C03663=1150.971,190.773,-61.352,-178.173,7.203,148.817
C03664=1150.967,191.022,-61.376,-178.171,7.205,148.817
C03665=1150.962,191.271,-61.399,-178.168,7.208,148.817
C03666=1150.958,191.521,-61.423,-178.165,7.210,148.817
C03667=1150.954,191.769,-61.447,-178.162,7.213,148.816
C03668=1150.949,192.018,-61.470,-178.160,7.214,148.816
C03669=1150.944,192.267,-61.493,-178.157,7.217,148.816
C03670=1150.940,192.516,-61.518,-178.154,7.219,148.816
C03671=1150.935,192.765,-61.541,-178.151,7.222,148.815
C03672=1150.931,193.013,-61.565,-178.149,7.224,148.815
C03673=1150.926,193.262,-61.588,-178.145,7.226,148.815
C03674=1150.921,193.511,-61.612,-178.143,7.228,148.815
C03675=1150.917,193.759,-61.636,-178.140,7.231,148.814
C03676=1150.912,194.008,-61.659,-178.138,7.233,148.814
C03677=1150.907,194.257,-61.684,-178.134,7.235,148.814
C03678=1150.902,194.506,-61.707,-178.132,7.238,148.814
C03679=1150.898,194.755,-61.731,-178.129,7.240,148.813
C03680=1150.893,195.004,-61.755,-178.127,7.242,148.813
C03681=1150.889,195.252,-61.779,-178.123,7.245,148.813
C03682=1150.884,195.501,-61.802,-178.121,7.247,148.813
C03683=1150.880,195.750,-61.826,-178.118,7.249,148.812
C03684=1150.876,195.999,-61.850,-178.115,7.251,148.812
C03685=1150.871,196.248,-61.874,-178.112,7.254,148.812
C03686=1150.866,196.497,-61.898,-178.110,7.256,148.812
C03687=1150.862,196.745,-61.922,-178.107,7.259,148.812
C03688=1150.857,196.994,-61.945,-178.104,7.261,148.811
C03689=1150.852,197.243,-61.969,-178.101,7.263,148.811
C03690=1150.848,197.491,-61.993,-178.098,7.266,148.811
C03691=1150.843,197.741,-62.018,-178.096,7.268,148.811
C03692=1150.839,197.990,-62.042,-178.093,7.271,148.810
C03693=1150.834,198.238,-62.066,-178.090,7.273,148.810
C03694=1150.830,198.487,-62.089,-178.087,7.275,148.810
C03695=1150.825,198.736,-62.113,-178.085,7.277,148.810
C03696=1150.820,198.984,-62.138,-178.082,7.280,148.809
C03697=1150.816,199.234,-62.162,-178.079,7.282,148.809
C03698=1150.812,199.482,-62.186,-178.076,7.285,148.809
C03699=1150.807,199.731,-62.210,-178.074,7.287,148.809
C03700=1150.802,199.980,-62.235,-178.071,7.289,148.808
C03701=1150.797,200.229,-62.258,-178.068,7.292,148.808
C03702=1150.794,200.478,-62.282,-178.065,7.294,148.808
C03703=1150.789,200.726,-62.307,-178.062,7.297,148.808
C03704=1150.784,200.975,-62.331,-178.060,7.299,148.808
C03705=1150.779,201.224,-62.354,-178.057,7.302,148.807
C03706=1150.775,201.472,-62.379,-178.054,7.303,148.807
C03707=1150.770,201.722,-62.404,-178.052,7.306,148.807
C03708=1150.766,201.970,-62.428,-178.049,7.308,148.807
C03709=1150.762,202.219,-62.452,-178.046,7.311,148.807
C03710=1150.757,202.467,-62.476,-178.043,7.314,148.806
C03711=1150.753,202.716,-62.501,-178.041,7.316,148.806
C03712=1150.748,202.965,-62.524,-178.038,7.319,148.806
C03713=1150.743,203.214,-62.549,-178.035,7.320,148.806
C03714=1150.739,203.463,-62.573,-178.032,7.323,148.805
C03715=1150.734,203.712,-62.598,-178.030,7.325,148.805
C03716=1150.730,203.960,-62.622,-178.027,7.328,148.805
C03717=1150.725,204.209,-62.646,-178.024,7.330,148.805
C03718=1150.721,204.458,-62.671,-178.021,7.333,148.805
C03719=1150.716,204.707,-62.695,-178.018,7.335,148.804
C03720=1150.711,204.955,-62.720,-178.016,7.337,148.804
C03721=1150.707,205.204,-62.744,-178.013,7.340,148.804
C03722=1150.702,205.453,-62.769,-178.010,7.343,148.804
C03723=1150.698,205.702,-62.793,-178.008,7.345,148.804
C03724=1150.693,205.950,-62.818,-178.004,7.347,148.803
C03725=1150.689,206.199,-62.842,-178.002,7.349,148.803
C03726=1150.684,206.448,-62.867,-177.999,7.352,148.803
C03727=1150.679,206.697,-62.891,-177.996,7.355,148.803
C03728=1150.675,206.946,-62.916,-177.993,7.357,148.802
C03729=1150.670,207.194,-62.940,-177.991,7.360,148.802
C03730=1150.666,207.443,-62.965,-177.988,7.362,148.802
C03731=1150.662,207.692,-62.990,-177.985,7.364,148.802
C03732=1150.657,207.940,-63.015,-177.982,7.367,148.802
C03733=1150.652,208.189,-63.039,-177.980,7.369,148.801
C03734=1150.648,208.438,-63.064,-177.977,7.372,148.801
C03735=1150.643,208.687,-63.088,-177.974,7.374,148.801
C03736=1150.639,208.936,-63.113,-177.971,7.377,148.801
C03737=1150.634,209.184,-63.138,-177.969,7.379,148.801
C03738=1150.629,209.454,-63.165,-177.965,7.382,148.800
C03739=1150.624,209.725,-63.192,-177.963,7.385,148.800
C03740=1150.619,209.995,-63.219,-177.960,7.387,148.800
C03741=1150.615,210.266,-63.246,-177.957,7.390,148.800
C03742=1150.610,210.515,-63.270,-177.954,7.392,148.800
C03743=1150.606,210.764,-63.295,-177.951,7.395,148.799
C03744=1150.601,211.013,-63.319,-177.948,7.397,148.799
C03745=1150.597,211.261,-63.345,-177.946,7.400,148.799
C03746=1150.592,211.510,-63.369,-177.943,7.403,148.799
C03747=1150.587,211.759,-63.394,-177.940,7.405,148.799
C03748=1150.583,212.007,-63.419,-177.937,7.407,148.798
C03749=1150.578,212.256,-63.444,-177.935,7.409,148.798
C03750=1150.574,212.505,-63.469,-177.932,7.412,148.798
C03751=1150.569,212.753,-63.494,-177.929,7.415,148.798
C03752=1150.565,213.003,-63.519,-177.926,7.417,148.798
C03753=1150.560,213.251,-63.544,-177.924,7.420,148.797
C03754=1150.556,213.500,-63.569,-177.921,7.423,148.797
C03755=1150.552,213.748,-63.594,-177.918,7.424,148.797
C03756=1150.547,213.997,-63.619,-177.915,7.427,148.797
C03757=1150.542,214.246,-63.644,-177.912,7.430,148.797
C03758=1150.538,214.495,-63.669,-177.910,7.432,148.797
C03759=1150.533,214.743,-63.693,-177.907,7.435,148.796
C03760=1150.529,214.992,-63.719,-177.904,7.437,148.796
C03761=1150.524,215.241,-63.744,-177.902,7.440,148.796
C03762=1150.520,215.490,-63.770,-177.899,7.443,148.796
C03763=1150.515,215.738,-63.794,-177.895,7.445,148.796
C03764=1150.511,215.987,-63.819,-177.893,7.447,148.795
C03765=1150.506,216.235,-63.845,-177.890,7.450,148.795
C03766=1150.502,216.484,-63.870,-177.887,7.453,148.795
C03767=1150.497,216.732,-63.895,-177.885,7.455,148.795
C03768=1150.492,216.982,-63.920,-177.882,7.458,148.795
C03769=1150.488,217.230,-63.945,-177.879,7.460,148.795
C03770=1150.484,217.478,-63.971,-177.877,7.462,148.794
C03771=1150.480,217.728,-63.996,-177.874,7.465,148.794
C03772=1150.475,217.976,-64.021,-177.871,7.468,148.794
C03773=1150.471,218.225,-64.047,-177.868,7.470,148.794
C03774=1150.465,218.474,-64.072,-177.866,7.473,148.794
C03775=1150.461,218.722,-64.097,-177.862,7.476,148.793
C03776=1150.457,218.971,-64.123,-177.860,7.478,148.793
C03777=1150.452,219.220,-64.148,-177.857,7.481,148.793
C03778=1150.448,219.468,-64.173,-177.855,7.483,148.793
C03779=1150.444,219.716,-64.198,-177.851,7.486,148.793
C03780=1150.439,219.965,-64.224,-177.849,7.488,148.793
C03781=1150.435,220.215,-64.249,-177.846,7.491,148.793
C03782=1150.430,220.463,-64.275,-177.843,7.494,148.792
C03783=1150.426,220.712,-64.300,-177.840,7.497,148.792
C03784=1150.421,220.960,-64.326,-177.838,7.499,148.792
C03785=1150.417,221.209,-64.351,-177.835,7.501,148.792
C03786=1150.412,221.458,-64.376,-177.832,7.504,148.792
C03787=1150.407,221.706,-64.402,-177.830,7.506,148.792
C03788=1150.403,221.955,-64.428,-177.827,7.509,148.792
C03789=1150.399,222.204,-64.453,-177.824,7.512,148.791
C03790=1150.394,222.452,-64.479,-177.821,7.515,148.791
C03791=1150.390,222.701,-64.504,-177.819,7.517,148.791
C03792=1150.386,222.949,-64.530,-177.816,7.519,148.791
C03793=1150.381,223.197,-64.556,-177.813,7.522,148.791
C03794=1150.377,223.446,-64.581,-177.811,7.524,148.790
C03795=1150.372,223.695,-64.607,-177.808,7.527,148.790
C03796=1150.367,223.944,-64.633,-177.805,7.530,148.790
C03797=1150.362,224.193,-64.658,-177.802,7.533,148.790
C03798=1150.358,224.442,-64.684,-177.800,7.535,148.790
C03799=1150.354,224.691,-64.710,-177.797,7.538,148.790
C03800=1150.349,224.939,-64.735,-177.793,7.540,148.789
C03801=1150.345,225.187,-64.761,-177.791,7.543,148.789
C03802=1150.341,225.436,-64.787,-177.788,7.545,148.789
C03803=1150.337,225.684,-64.813,-177.786,7.548,148.789
C03804=1150.332,225.933,-64.838,-177.782,7.551,148.789
C03805=1150.327,226.182,-64.865,-177.780,7.554,148.789
C03806=1150.323,226.430,-64.890,-177.777,7.556,148.789
C03807=1150.318,226.679,-64.916,-177.775,7.559,148.789
C03808=1150.314,226.927,-64.942,-177.771,7.562,148.788
C03809=1150.309,227.176,-64.967,-177.769,7.564,148.788
C03810=1150.304,227.425,-64.994,-177.766,7.567,148.788
C03811=1150.300,227.673,-65.020,-177.764,7.569,148.788
C03812=1150.296,227.922,-65.046,-177.760,7.572,148.788
C03813=1150.291,228.170,-65.071,-177.758,7.575,148.788
C03814=1150.287,228.419,-65.097,-177.755,7.578,148.788
C03815=1150.282,228.668,-65.123,-177.753,7.580,148.787
C03816=1150.278,228.917,-65.149,-177.750,7.583,148.787
C03817=1150.273,229.165,-65.175,-177.747,7.586,148.787
C03818=1150.269,229.413,-65.201,-177.744,7.588,148.787
C03819=1150.264,229.663,-65.227,-177.742,7.591,148.787
C03820=1150.260,229.911,-65.254,-177.739,7.593,148.787
C03821=1150.256,230.160,-65.280,-177.736,7.596,148.786
C03822=1150.251,230.409,-65.306,-177.733,7.599,148.786
C03823=1150.246,230.657,-65.331,-177.730,7.602,148.786
C03824=1150.242,230.905,-65.358,-177.728,7.604,148.786
C03825=1150.237,231.154,-65.384,-177.725,7.607,148.786
C03826=1150.233,231.403,-65.410,-177.722,7.610,148.786
C03827=1150.229,231.651,-65.436,-177.719,7.612,148.786
C03828=1150.224,231.900,-65.463,-177.716,7.615,148.786
C03829=1150.220,232.148,-65.489,-177.714,7.618,148.785
C03830=1150.216,232.396,-65.514,-177.711,7.620,148.785
C03831=1150.211,232.646,-65.541,-177.708,7.623,148.785
C03832=1150.207,232.894,-65.567,-177.705,7.626,148.785
C03833=1150.202,233.143,-65.594,-177.702,7.629,148.785
C03834=1150.198,233.391,-65.620,-177.700,7.631,148.785
C03835=1150.194,233.640,-65.646,-177.697,7.634,148.785
C03836=1150.189,233.888,-65.673,-177.695,7.637,148.785
C03837=1150.185,234.137,-65.699,-177.691,7.639,148.784
C03838=1150.180,234.386,-65.726,-177.688,7.642,148.784
C03839=1150.176,234.634,-65.751,-177.686,7.644,148.784
C03840=1150.171,234.882,-65.778,-177.684,7.647,148.784
C03841=1150.166,235.131,-65.804,-177.681,7.650,148.784
C03842=1150.162,235.403,-65.834,-177.678,7.653,148.784
C03843=1150.157,235.675,-65.862,-177.675,7.656,148.784
C03844=1150.152,235.947,-65.891,-177.671,7.660,148.784
C03845=1150.148,236.218,-65.920,-177.669,7.663,148.784
C03846=1150.143,236.467,-65.947,-177.666,7.665,148.783
C03847=1150.139,236.715,-65.973,-177.663,7.667,148.783
C03848=1150.134,236.964,-66.000,-177.660,7.670,148.783
C03849=1150.130,237.213,-66.025,-177.658,7.673,148.783
C03850=1150.125,237.461,-66.052,-177.655,7.676,148.783
C03851=1150.121,237.710,-66.080,-177.652,7.679,148.783
C03852=1150.117,237.958,-66.106,-177.649,7.682,148.783
C03853=1150.112,238.207,-66.132,-177.646,7.685,148.783
C03854=1150.108,238.455,-66.159,-177.644,7.687,148.782
C03855=1150.103,238.704,-66.186,-177.641,7.689,148.782
C03856=1150.099,238.952,-66.212,-177.638,7.692,148.782
C03857=1150.094,239.201,-66.239,-177.635,7.695,148.782
C03858=1150.090,239.449,-66.266,-177.633,7.698,148.782
C03859=1150.086,239.698,-66.292,-177.630,7.701,148.782
C03860=1150.081,239.946,-66.319,-177.628,7.703,148.782
C03861=1150.076,240.195,-66.346,-177.625,7.706,148.782
C03862=1150.072,240.443,-66.372,-177.622,7.709,148.782
C03863=1150.067,240.692,-66.399,-177.619,7.712,148.781
C03864=1150.063,240.940,-66.426,-177.616,7.715,148.781
C03865=1150.059,241.189,-66.453,-177.613,7.718,148.781
C03866=1150.054,241.437,-66.480,-177.610,7.721,148.781
C03867=1150.050,241.686,-66.507,-177.608,7.723,148.781
C03868=1150.046,241.935,-66.534,-177.605,7.726,148.781
C03869=1150.041,242.184,-66.560,-177.603,7.728,148.781
C03870=1150.037,242.432,-66.587,-177.600,7.731,148.781
C03871=1150.033,242.680,-66.614,-177.597,7.734,148.781
C03872=1150.028,242.929,-66.641,-177.594,7.737,148.781
C03873=1150.023,243.177,-66.668,-177.591,7.740,148.780
C03874=1150.019,243.426,-66.695,-177.588,7.743,148.780
C03875=1150.015,243.674,-66.721,-177.585,7.746,148.780
C03876=1150.011,243.923,-66.749,-177.583,7.748,148.780
C03877=1150.006,244.172,-66.776,-177.580,7.751,148.780
C03878=1150.001,244.420,-66.803,-177.578,7.754,148.780
C03879=1149.997,244.669,-66.830,-177.575,7.757,148.780
C03880=1149.993,244.916,-66.857,-177.572,7.760,148.780
C03881=1149.988,245.165,-66.884,-177.569,7.763,148.780
C03882=1149.984,245.413,-66.911,-177.567,7.765,148.780
C03883=1149.980,245.662,-66.939,-177.564,7.768,148.780
C03884=1149.975,245.911,-66.966,-177.561,7.771,148.780
C03885=1149.970,246.159,-66.993,-177.559,7.773,148.779
C03886=1149.967,246.408,-67.019,-177.556,7.776,148.779
C03887=1149.962,246.656,-67.046,-177.553,7.779,148.779
C03888=1149.958,246.904,-67.074,-177.550,7.782,148.779
C03889=1149.953,247.153,-67.101,-177.547,7.785,148.779
C03890=1149.949,247.402,-67.128,-177.544,7.788,148.779
C03891=1149.944,247.650,-67.155,-177.542,7.791,148.779
C03892=1149.940,247.899,-67.183,-177.539,7.794,148.779
C03893=1149.936,248.147,-67.211,-177.536,7.797,148.779
C03894=1149.931,248.396,-67.238,-177.533,7.799,148.779
C03895=1149.926,248.644,-67.265,-177.531,7.802,148.778
C03896=1149.923,248.892,-67.291,-177.528,7.804,148.778
C03897=1149.918,249.140,-67.319,-177.526,7.807,148.778
C03898=1149.914,249.389,-67.346,-177.523,7.810,148.778
C03899=1149.909,249.638,-67.374,-177.520,7.813,148.778
C03900=1149.905,249.886,-67.401,-177.517,7.816,148.778
C03901=1149.900,250.134,-67.428,-177.514,7.819,148.778
C03902=1149.896,250.384,-67.456,-177.512,7.822,148.778
C03903=1149.892,250.631,-67.484,-177.509,7.825,148.778
C03904=1149.887,250.880,-67.511,-177.506,7.828,148.778
C03905=1149.884,251.128,-67.539,-177.503,7.831,148.778
C03906=1149.879,251.377,-67.566,-177.500,7.834,148.778
C03907=1149.875,251.625,-67.594,-177.498,7.837,148.778
C03908=1149.870,251.873,-67.621,-177.495,7.840,148.778
C03909=1149.865,252.123,-67.649,-177.493,7.842,148.777
C03910=1149.861,252.371,-67.676,-177.490,7.845,148.777
C03911=1149.856,252.619,-67.704,-177.487,7.848,148.777
C03912=1149.852,252.868,-67.732,-177.484,7.851,148.777
C03913=1149.848,253.116,-67.759,-177.482,7.854,148.777
C03914=1149.843,253.364,-67.787,-177.479,7.856,148.777
C03915=1149.839,253.613,-67.814,-177.476,7.859,148.777
C03916=1149.835,253.861,-67.842,-177.473,7.862,148.777
C03917=1149.831,254.109,-67.870,-177.470,7.865,148.777
C03918=1149.827,254.358,-67.897,-177.468,7.868,148.777
C03919=1149.822,254.607,-67.925,-177.465,7.871,148.777
C03920=1149.817,254.855,-67.952,-177.462,7.874,148.777
C03921=1149.813,255.104,-67.981,-177.459,7.877,148.777
C03922=1149.809,255.351,-68.008,-177.457,7.880,148.777
C03923=1149.805,255.601,-68.036,-177.454,7.883,148.777
C03924=1149.800,255.849,-68.064,-177.451,7.886,148.777
C03925=1149.795,256.097,-68.092,-177.449,7.889,148.777
C03926=1149.791,256.346,-68.119,-177.446,7.892,148.777
C03927=1149.787,256.594,-68.147,-177.443,7.895,148.776
C03928=1149.783,256.842,-68.175,-177.440,7.898,148.776
C03929=1149.778,257.091,-68.203,-177.438,7.901,148.776
C03930=1149.773,257.339,-68.231,-177.435,7.904,148.776
C03931=1149.770,257.588,-68.259,-177.433,7.906,148.776
C03932=1149.765,257.835,-68.287,-177.430,7.909,148.776
C03933=1149.760,258.085,-68.315,-177.427,7.912,148.776
C03934=1149.756,258.333,-68.342,-177.424,7.915,148.776
C03935=1149.752,258.581,-68.371,-177.421,7.918,148.776
C03936=1149.748,258.829,-68.398,-177.419,7.921,148.776
C03937=1149.743,259.078,-68.427,-177.416,7.923,148.776
C03938=1149.739,259.326,-68.455,-177.414,7.927,148.776
C03939=1149.735,259.575,-68.482,-177.411,7.930,148.776
C03940=1149.730,259.823,-68.511,-177.408,7.933,148.776
C03941=1149.726,260.071,-68.538,-177.405,7.936,148.776
C03942=1149.722,260.320,-68.567,-177.402,7.938,148.776
C03943=1149.717,260.568,-68.595,-177.400,7.941,148.776
C03944=1149.713,260.817,-68.623,-177.397,7.944,148.776
C03945=1149.709,261.065,-68.651,-177.394,7.947,148.776
C03946=1149.703,261.338,-68.682,-177.391,7.951,148.776
C03947=1149.699,261.612,-68.713,-177.388,7.954,148.775
C03948=1149.695,261.886,-68.744,-177.385,7.957,148.775
C03949=1149.690,262.159,-68.776,-177.382,7.961,148.775
C03950=1149.685,262.406,-68.804,-177.379,7.964,148.775
C03951=1149.681,262.655,-68.832,-177.377,7.967,148.775
C03952=1149.676,262.903,-68.860,-177.374,7.970,148.775
C03953=1149.673,263.152,-68.888,-177.371,7.973,148.775
C03954=1149.667,263.400,-68.917,-177.368,7.976,148.775
C03955=1149.664,263.649,-68.945,-177.366,7.979,148.775
C03956=1149.659,263.897,-68.973,-177.363,7.982,148.775
C03957=1149.655,264.145,-69.001,-177.360,7.984,148.775
C03958=1149.650,264.394,-69.030,-177.357,7.987,148.775
C03959=1149.646,264.642,-69.058,-177.355,7.991,148.775
C03960=1149.642,264.890,-69.087,-177.352,7.994,148.775
C03961=1149.638,265.138,-69.115,-177.349,7.997,148.775
C03962=1149.633,265.387,-69.144,-177.347,7.999,148.775
C03963=1149.629,265.636,-69.172,-177.344,8.002,148.775
C03964=1149.624,265.884,-69.200,-177.341,8.005,148.775
C03965=1149.621,266.132,-69.229,-177.339,8.009,148.775
C03966=1149.616,266.380,-69.258,-177.336,8.012,148.775
C03967=1149.611,266.629,-69.286,-177.333,8.014,148.775
C03968=1149.607,266.878,-69.314,-177.330,8.017,148.775
C03969=1149.603,267.125,-69.343,-177.328,8.020,148.775
C03970=1149.599,267.374,-69.372,-177.325,8.023,148.775
C03971=1149.594,267.622,-69.400,-177.323,8.027,148.775
C03972=1149.590,267.870,-69.429,-177.320,8.029,148.775
C03973=1149.586,268.119,-69.458,-177.317,8.032,148.775
C03974=1149.581,268.367,-69.486,-177.314,8.035,148.775
C03975=1149.577,268.615,-69.515,-177.311,8.038,148.775
C03976=1149.573,268.864,-69.544,-177.309,8.042,148.775
C03977=1149.568,269.112,-69.572,-177.306,8.045,148.775
C03978=1149.564,269.360,-69.601,-177.303,8.048,148.775
C03979=1149.560,269.609,-69.630,-177.300,8.051,148.775
C03980=1149.555,269.856,-69.659,-177.297,8.054,148.775
C03981=1149.551,270.105,-69.687,-177.295,8.057,148.775
C03982=1149.547,270.354,-69.715,-177.292,8.060,148.775
C03983=1149.543,270.602,-69.745,-177.290,8.063,148.775
C03984=1149.538,270.850,-69.773,-177.287,8.066,148.775
C03985=1149.534,271.098,-69.802,-177.284,8.069,148.775
C03986=1149.530,271.347,-69.831,-177.282,8.072,148.775
C03987=1149.525,271.595,-69.860,-177.279,8.075,148.775
C03988=1149.520,271.844,-69.889,-177.276,8.078,148.775
C03989=1149.517,272.091,-69.918,-177.273,8.081,148.775
C03990=1149.513,272.340,-69.947,-177.271,8.084,148.775
C03991=1149.508,272.588,-69.975,-177.268,8.087,148.775
C03992=1149.503,272.836,-70.005,-177.265,8.090,148.775
C03993=1149.499,273.085,-70.034,-177.262,8.094,148.775
C03994=1149.496,273.333,-70.062,-177.260,8.097,148.775
C03995=1149.491,273.581,-70.092,-177.257,8.100,148.775
C03996=1149.486,273.830,-70.120,-177.254,8.103,148.775
C03997=1149.482,274.078,-70.150,-177.251,8.106,148.775
C03998=1149.478,274.326,-70.179,-177.249,8.109,148.775
C03999=1149.473,274.575,-70.208,-177.246,8.112,148.775
C04000=1149.469,274.822,-70.236,-177.244,8.115,148.775
C04001=1149.465,275.070,-70.266,-177.241,8.118,148.775
C04002=1149.461,275.319,-70.295,-177.238,8.122,148.775
C04003=1149.457,275.568,-70.324,-177.236,8.125,148.775
C04004=1149.452,275.816,-70.354,-177.233,8.127,148.775
C04005=1149.448,276.064,-70.383,-177.230,8.130,148.775
C04006=1149.443,276.312,-70.412,-177.227,8.134,148.775
C04007=1149.439,276.561,-70.441,-177.224,8.137,148.775
C04008=1149.435,276.809,-70.470,-177.222,8.140,148.775
C04009=1149.431,277.057,-70.499,-177.219,8.144,148.775
C04010=1149.427,277.305,-70.529,-177.217,8.147,148.775
C04011=1149.423,277.553,-70.558,-177.214,8.149,148.775
C04012=1149.418,277.801,-70.587,-177.212,8.153,148.775
C04013=1149.414,278.050,-70.616,-177.209,8.156,148.775
C04014=1149.409,278.298,-70.645,-177.206,8.159,148.775
C04015=1149.405,278.546,-70.675,-177.203,8.162,148.775
C04016=1149.401,278.795,-70.704,-177.200,8.166,148.775
C04017=1149.397,279.043,-70.734,-177.198,8.169,148.775
C04018=1149.393,279.291,-70.763,-177.195,8.172,148.775
C04019=1149.389,279.539,-70.793,-177.192,8.175,148.775
C04020=1149.384,279.788,-70.822,-177.190,8.178,148.775
C04021=1149.380,280.036,-70.851,-177.187,8.181,148.775
C04022=1149.375,280.284,-70.881,-177.185,8.184,148.775
C04023=1149.371,280.532,-70.910,-177.182,8.187,148.775
C04024=1149.366,280.780,-70.940,-177.179,8.190,148.775
C04025=1149.362,281.029,-70.970,-177.176,8.194,148.775
C04026=1149.358,281.277,-70.999,-177.173,8.197,148.775
C04027=1149.354,281.525,-71.028,-177.171,8.200,148.775
C04028=1149.350,281.773,-71.058,-177.168,8.203,148.775
C04029=1149.345,282.022,-71.087,-177.165,8.206,148.775
C04030=1149.342,282.269,-71.118,-177.163,8.209,148.775
C04031=1149.337,282.518,-71.147,-177.160,8.212,148.775
C04032=1149.332,282.766,-71.177,-177.158,8.215,148.775
C04033=1149.328,283.014,-71.206,-177.155,8.219,148.776
C04034=1149.324,283.263,-71.236,-177.152,8.222,148.776
C04035=1149.320,283.511,-71.265,-177.149,8.225,148.776
C04036=1149.316,283.759,-71.295,-177.147,8.228,148.776
C04037=1149.312,284.007,-71.325,-177.144,8.231,148.776
C04038=1149.307,284.255,-71.355,-177.142,8.235,148.776
C04039=1149.303,284.504,-71.384,-177.139,8.238,148.776
C04040=1149.299,284.752,-71.414,-177.136,8.241,148.776
C04041=1149.295,285.000,-71.444,-177.133,8.245,148.776
C04042=1149.290,285.248,-71.474,-177.130,8.248,148.776
C04043=1149.286,285.497,-71.504,-177.128,8.251,148.776
C04044=1149.282,285.744,-71.534,-177.125,8.254,148.776
C04045=1149.277,285.992,-71.563,-177.123,8.257,148.776
C04046=1149.273,286.241,-71.593,-177.120,8.260,148.776
C04047=1149.269,286.489,-71.623,-177.117,8.264,148.776
C04048=1149.265,286.737,-71.653,-177.115,8.267,148.776
C04049=1149.260,286.985,-71.682,-177.112,8.270,148.776
C04050=1149.256,287.261,-71.717,-177.109,8.273,148.776
C04051=1149.251,287.536,-71.749,-177.106,8.277,148.776
C04052=1149.246,287.811,-71.783,-177.103,8.281,148.776
C04053=1149.241,288.086,-71.816,-177.100,8.284,148.776
C04054=1149.238,288.335,-71.846,-177.097,8.288,148.777
C04055=1149.233,288.583,-71.876,-177.094,8.291,148.777
C04056=1149.229,288.831,-71.906,-177.092,8.294,148.777
C04057=1149.224,289.079,-71.937,-177.089,8.297,148.777
C04058=1149.220,289.327,-71.966,-177.087,8.300,148.777
C04059=1149.216,289.575,-71.996,-177.084,8.303,148.777
C04060=1149.211,289.824,-72.026,-177.081,8.307,148.777
C04061=1149.207,290.071,-72.057,-177.078,8.310,148.777
C04062=1149.203,290.320,-72.087,-177.076,8.313,148.777
C04063=1149.199,290.568,-72.117,-177.073,8.316,148.777
C04064=1149.195,290.816,-72.147,-177.071,8.319,148.777
C04065=1149.191,291.064,-72.177,-177.068,8.323,148.777
C04066=1149.187,291.312,-72.207,-177.065,8.326,148.777
C04067=1149.182,291.561,-72.238,-177.063,8.330,148.777
C04068=1149.178,291.808,-72.268,-177.060,8.333,148.777
C04069=1149.174,292.057,-72.299,-177.058,8.336,148.778
C04070=1149.170,292.305,-72.328,-177.055,8.339,148.777
C04071=1149.165,292.553,-72.359,-177.052,8.343,148.778
C04072=1149.161,292.801,-72.389,-177.049,8.346,148.778
C04073=1149.156,293.049,-72.419,-177.047,8.349,148.778
C04074=1149.153,293.298,-72.450,-177.044,8.352,148.778
C04075=1149.148,293.546,-72.481,-177.042,8.355,148.778
C04076=1149.144,293.793,-72.511,-177.038,8.359,148.778
C04077=1149.140,294.042,-72.541,-177.036,8.362,148.778
C04078=1149.136,294.290,-72.571,-177.033,8.365,148.778
C04079=1149.132,294.538,-72.602,-177.031,8.369,148.778
C04080=1149.128,294.786,-72.632,-177.029,8.372,148.778
C04081=1149.123,295.034,-72.663,-177.025,8.376,148.778
C04082=1149.119,295.282,-72.694,-177.023,8.379,148.779
C04083=1149.115,295.531,-72.724,-177.020,8.382,148.779
C04084=1149.110,295.779,-72.754,-177.018,8.385,148.779
C04085=1149.106,296.026,-72.785,-177.015,8.388,148.779
C04086=1149.102,296.275,-72.816,-177.012,8.392,148.779
C04087=1149.098,296.523,-72.846,-177.009,8.395,148.779
C04088=1149.094,296.771,-72.877,-177.007,8.398,148.779
C04089=1149.089,297.019,-72.907,-177.004,8.401,148.779
C04090=1149.085,297.267,-72.938,-177.002,8.404,148.779
C04091=1149.081,297.515,-72.969,-176.999,8.409,148.779
C04092=1149.077,297.763,-72.999,-176.996,8.412,148.779
C04093=1149.073,298.011,-73.031,-176.994,8.415,148.780
C04094=1149.069,298.259,-73.061,-176.991,8.418,148.780
C04095=1149.064,298.507,-73.091,-176.988,8.422,148.780
C04096=1149.060,298.756,-73.123,-176.986,8.425,148.780
C04097=1149.056,299.003,-73.153,-176.983,8.428,148.780
C04098=1149.052,299.251,-73.184,-176.981,8.431,148.780
C04099=1149.048,299.500,-73.215,-176.978,8.435,148.780
C04100=1149.043,299.748,-73.245,-176.975,8.438,148.780
C04101=1149.039,299.996,-73.276,-176.972,8.441,148.780
C04102=1149.035,300.244,-73.307,-176.970,8.445,148.780
C04103=1149.031,300.492,-73.338,-176.968,8.448,148.781
C04104=1149.026,300.740,-73.369,-176.964,8.452,148.781
C04105=1149.022,300.988,-73.400,-176.962,8.455,148.781
C04106=1149.019,301.236,-73.430,-176.959,8.458,148.781
C04107=1149.014,301.484,-73.461,-176.957,8.461,148.781
C04108=1149.010,301.732,-73.492,-176.954,8.465,148.781
C04109=1149.006,301.980,-73.524,-176.951,8.468,148.781
C04110=1149.002,302.228,-73.555,-176.949,8.471,148.781
C04111=1148.997,302.476,-73.586,-176.947,8.475,148.781
C04112=1148.993,302.724,-73.616,-176.943,8.478,148.781
C04113=1148.989,302.972,-73.648,-176.941,8.482,148.782
C04114=1148.985,303.220,-73.678,-176.939,8.485,148.782
C04115=1148.981,303.469,-73.709,-176.936,8.488,148.782
C04116=1148.976,303.716,-73.741,-176.933,8.492,148.782
C04117=1148.972,303.964,-73.772,-176.931,8.495,148.782
C04118=1148.968,304.213,-73.803,-176.928,8.498,148.782
C04119=1148.964,304.460,-73.834,-176.925,8.502,148.782
C04120=1148.960,304.709,-73.865,-176.923,8.506,148.783
C04121=1148.955,304.957,-73.896,-176.920,8.508,148.783
C04122=1148.951,305.205,-73.928,-176.918,8.512,148.783
C04123=1148.947,305.453,-73.959,-176.915,8.516,148.783
C04124=1148.943,305.701,-73.991,-176.912,8.519,148.783
C04125=1148.938,305.949,-74.021,-176.910,8.522,148.783
C04126=1148.935,306.197,-74.053,-176.907,8.525,148.783
C04127=1148.930,306.445,-74.084,-176.904,8.529,148.783
C04128=1148.926,306.693,-74.116,-176.902,8.532,148.783
C04129=1148.922,306.941,-74.147,-176.899,8.536,148.784
C04130=1148.918,307.189,-74.178,-176.896,8.539,148.784
C04131=1148.913,307.437,-74.209,-176.894,8.543,148.784
C04132=1148.910,307.685,-74.241,-176.891,8.546,148.784
C04133=1148.905,307.933,-74.272,-176.889,8.549,148.784
C04134=1148.901,308.181,-74.304,-176.886,8.553,148.784
C04135=1148.897,308.429,-74.334,-176.883,8.556,148.784
C04136=1148.893,308.677,-74.366,-176.881,8.560,148.785
C04137=1148.889,308.924,-74.398,-176.878,8.563,148.785
C04138=1148.885,309.173,-74.429,-176.875,8.567,148.785
C04139=1148.880,309.420,-74.460,-176.873,8.570,148.785
C04140=1148.877,309.668,-74.492,-176.871,8.573,148.785
C04141=1148.871,309.916,-74.524,-176.867,8.577,148.785
C04142=1148.868,310.164,-74.555,-176.865,8.580,148.785
C04143=1148.864,310.412,-74.587,-176.863,8.583,148.786
C04144=1148.859,310.660,-74.618,-176.860,8.587,148.786
C04145=1148.856,310.908,-74.650,-176.857,8.590,148.786
C04146=1148.851,311.156,-74.681,-176.855,8.594,148.786
C04147=1148.848,311.404,-74.713,-176.852,8.598,148.786
C04148=1148.842,311.652,-74.745,-176.849,8.601,148.786
C04149=1148.838,311.900,-74.776,-176.847,8.604,148.786
C04150=1148.835,312.148,-74.808,-176.844,8.608,148.787
C04151=1148.830,312.395,-74.840,-176.841,8.611,148.787
C04152=1148.827,312.643,-74.872,-176.839,8.615,148.787
C04153=1148.822,312.892,-74.904,-176.837,8.618,148.787
C04154=1148.817,313.169,-74.939,-176.833,8.622,148.787
C04155=1148.813,313.447,-74.974,-176.831,8.626,148.787
C04156=1148.808,313.724,-75.010,-176.828,8.630,148.788
C04157=1148.803,314.002,-75.046,-176.825,8.634,148.788
C04158=1148.800,314.250,-75.078,-176.822,8.637,148.788
C04159=1148.795,314.498,-75.109,-176.819,8.641,148.788
C04160=1148.791,314.746,-75.142,-176.817,8.644,148.788
C04161=1148.787,314.994,-75.174,-176.814,8.648,148.788
C04162=1148.783,315.241,-75.205,-176.811,8.652,148.789
C04163=1148.779,315.489,-75.237,-176.809,8.655,148.789
C04164=1148.775,315.738,-75.269,-176.806,8.658,148.789
C04165=1148.770,315.985,-75.301,-176.803,8.662,148.789
C04166=1148.767,316.233,-75.333,-176.801,8.665,148.789
C04167=1148.762,316.481,-75.365,-176.799,8.668,148.789
C04168=1148.759,316.729,-75.397,-176.796,8.673,148.790
C04169=1148.754,316.977,-75.429,-176.794,8.676,148.790
C04170=1148.750,317.225,-75.461,-176.791,8.679,148.790
C04171=1148.746,317.473,-75.493,-176.788,8.683,148.790
C04172=1148.742,317.721,-75.525,-176.786,8.686,148.790
C04173=1148.737,317.969,-75.557,-176.783,8.689,148.790
C04174=1148.733,318.217,-75.590,-176.780,8.693,148.791
C04175=1148.730,318.465,-75.622,-176.778,8.697,148.791
C04176=1148.726,318.713,-75.653,-176.776,8.700,148.791
C04177=1148.721,318.960,-75.686,-176.773,8.704,148.791
C04178=1148.717,319.208,-75.717,-176.770,8.707,148.791
C04179=1148.713,319.456,-75.751,-176.768,8.710,148.791
C04180=1148.709,319.704,-75.782,-176.765,8.714,148.792
C04181=1148.705,319.952,-75.815,-176.762,8.718,148.792
C04182=1148.701,320.200,-75.846,-176.760,8.722,148.792
C04183=1148.696,320.447,-75.879,-176.757,8.725,148.792
C04184=1148.693,320.696,-75.911,-176.755,8.728,148.792
C04185=1148.688,320.944,-75.944,-176.752,8.732,148.793
C04186=1148.685,321.191,-75.976,-176.750,8.736,148.793
C04187=1148.680,321.439,-76.008,-176.747,8.739,148.793
C04188=1148.676,321.687,-76.040,-176.744,8.743,148.793
C04189=1148.672,321.935,-76.073,-176.742,8.746,148.793
C04190=1148.668,322.183,-76.105,-176.739,8.750,148.793
C04191=1148.664,322.431,-76.138,-176.736,8.753,148.794
C04192=1148.660,322.679,-76.170,-176.734,8.757,148.794
C04193=1148.656,322.927,-76.203,-176.731,8.761,148.794
C04194=1148.651,323.174,-76.235,-176.729,8.764,148.794
C04195=1148.647,323.422,-76.267,-176.727,8.767,148.794
C04196=1148.643,323.670,-76.300,-176.724,8.771,148.795
C04197=1148.640,323.918,-76.332,-176.721,8.775,148.795
C04198=1148.636,324.165,-76.365,-176.718,8.779,148.795
C04199=1148.631,324.414,-76.398,-176.716,8.782,148.795
C04200=1148.628,324.661,-76.430,-176.714,8.785,148.795
C04201=1148.623,324.910,-76.463,-176.711,8.789,148.796
C04202=1148.618,325.157,-76.496,-176.709,8.793,148.796
C04203=1148.615,325.405,-76.528,-176.706,8.797,148.796
C04204=1148.611,325.652,-76.561,-176.703,8.800,148.796
C04205=1148.607,325.900,-76.594,-176.701,8.803,148.797
C04206=1148.603,326.148,-76.626,-176.698,8.807,148.797
C04207=1148.599,326.396,-76.659,-176.696,8.811,148.797
C04208=1148.594,326.644,-76.691,-176.693,8.815,148.797
C04209=1148.591,326.892,-76.724,-176.691,8.818,148.797
C04210=1148.587,327.139,-76.757,-176.688,8.822,148.798
C04211=1148.582,327.388,-76.789,-176.685,8.825,148.798
C04212=1148.578,327.635,-76.823,-176.683,8.829,148.798
C04213=1148.575,327.883,-76.855,-176.680,8.833,148.798
C04214=1148.571,328.131,-76.888,-176.678,8.836,148.798
C04215=1148.566,328.379,-76.921,-176.675,8.840,148.799
C04216=1148.562,328.627,-76.954,-176.673,8.843,148.799
C04217=1148.558,328.874,-76.987,-176.670,8.846,148.799
C04218=1148.554,329.122,-77.020,-176.667,8.851,148.799
C04219=1148.550,329.370,-77.052,-176.665,8.854,148.799
C04220=1148.546,329.618,-77.085,-176.662,8.858,148.800
C04221=1148.542,329.866,-77.118,-176.660,8.861,148.800
C04222=1148.538,330.113,-77.152,-176.657,8.865,148.800
C04223=1148.533,330.361,-77.185,-176.654,8.869,148.800
C04224=1148.529,330.609,-77.218,-176.652,8.872,148.801
C04225=1148.526,330.856,-77.250,-176.649,8.876,148.801
C04226=1148.521,331.105,-77.283,-176.647,8.879,148.801
C04227=1148.517,331.352,-77.316,-176.644,8.883,148.801
C04228=1148.513,331.600,-77.349,-176.642,8.887,148.801
C04229=1148.509,331.848,-77.382,-176.639,8.891,148.802
C04230=1148.505,332.095,-77.416,-176.637,8.894,148.802
C04231=1148.501,332.343,-77.449,-176.634,8.898,148.802
C04232=1148.497,332.591,-77.482,-176.632,8.902,148.803
C04233=1148.492,332.839,-77.515,-176.629,8.905,148.803
C04234=1148.488,333.086,-77.548,-176.626,8.909,148.803
C04235=1148.484,333.334,-77.581,-176.624,8.912,148.803
C04236=1148.480,333.582,-77.614,-176.621,8.916,148.803
C04237=1148.476,333.830,-77.648,-176.619,8.920,148.804
C04238=1148.472,334.078,-77.681,-176.616,8.924,148.804
C04239=1148.469,334.325,-77.715,-176.614,8.927,148.804
C04240=1148.464,334.573,-77.748,-176.611,8.931,148.804
C04241=1148.460,334.821,-77.781,-176.609,8.935,148.805
C04242=1148.456,335.068,-77.814,-176.606,8.939,148.805
C04243=1148.452,335.316,-77.848,-176.604,8.942,148.805
C04244=1148.448,335.564,-77.881,-176.601,8.946,148.805
C04245=1148.444,335.811,-77.914,-176.598,8.949,148.806
C04246=1148.441,336.059,-77.948,-176.595,8.953,148.806
C04247=1148.436,336.307,-77.981,-176.593,8.957,148.806
C04248=1148.432,336.555,-78.014,-176.591,8.960,148.806
C04249=1148.428,336.802,-78.048,-176.588,8.964,148.807
C04250=1148.424,337.050,-78.082,-176.586,8.968,148.807
C04251=1148.420,337.297,-78.115,-176.583,8.972,148.807
C04252=1148.417,337.546,-78.148,-176.581,8.975,148.807
C04253=1148.412,337.794,-78.182,-176.578,8.979,148.808
C04254=1148.408,338.041,-78.216,-176.576,8.983,148.808
C04255=1148.404,338.289,-78.249,-176.573,8.987,148.808
C04256=1148.400,338.536,-78.282,-176.571,8.990,148.808
C04257=1148.396,338.784,-78.316,-176.568,8.994,148.809
C04258=1148.391,339.064,-78.354,-176.565,8.998,148.809
C04259=1148.387,339.344,-78.392,-176.562,9.003,148.809
C04260=1148.382,339.625,-78.431,-176.560,9.007,148.810
C04261=1148.377,339.905,-78.468,-176.557,9.011,148.810
C04262=1148.374,340.153,-78.502,-176.554,9.015,148.810
C04263=1148.369,340.401,-78.536,-176.551,9.018,148.810
C04264=1148.365,340.648,-78.570,-176.549,9.022,148.811
C04265=1148.361,340.896,-78.603,-176.547,9.026,148.811
C04266=1148.357,341.143,-78.637,-176.544,9.030,148.811
C04267=1148.353,341.392,-78.671,-176.541,9.033,148.811
C04268=1148.349,341.639,-78.705,-176.538,9.037,148.812
C04269=1148.345,341.887,-78.738,-176.537,9.041,148.812
C04270=1148.341,342.134,-78.772,-176.534,9.045,148.812
C04271=1148.337,342.382,-78.806,-176.531,9.048,148.812
C04272=1148.333,342.630,-78.840,-176.528,9.052,148.813
C04273=1148.329,342.877,-78.874,-176.527,9.056,148.813
C04274=1148.325,343.125,-78.908,-176.524,9.060,148.813
C04275=1148.321,343.372,-78.941,-176.521,9.063,148.814
C04276=1148.316,343.621,-78.975,-176.518,9.067,148.814
C04277=1148.313,343.868,-79.009,-176.516,9.071,148.814
C04278=1148.309,344.115,-79.043,-176.514,9.075,148.814
C04279=1148.305,344.363,-79.077,-176.511,9.079,148.815
C04280=1148.301,344.611,-79.111,-176.508,9.082,148.815
C04281=1148.297,344.859,-79.146,-176.506,9.087,148.815
C04282=1148.293,345.106,-79.180,-176.504,9.090,148.816
C04283=1148.289,345.354,-79.213,-176.501,9.094,148.816
C04284=1148.285,345.602,-79.248,-176.498,9.097,148.816
C04285=1148.281,345.849,-79.281,-176.496,9.102,148.817
C04286=1148.277,346.097,-79.316,-176.493,9.105,148.817
C04287=1148.273,346.345,-79.349,-176.491,9.109,148.817
C04288=1148.268,346.592,-79.384,-176.489,9.113,148.817
C04289=1148.265,346.840,-79.418,-176.486,9.117,148.818
C04290=1148.261,347.087,-79.453,-176.483,9.120,148.818
C04291=1148.257,347.334,-79.487,-176.480,9.124,148.818
C04292=1148.253,347.583,-79.521,-176.478,9.128,148.819
C04293=1148.249,347.830,-79.555,-176.476,9.132,148.819
C04294=1148.245,348.078,-79.589,-176.473,9.136,148.819
C04295=1148.241,348.325,-79.623,-176.471,9.139,148.819
C04296=1148.236,348.573,-79.658,-176.468,9.144,148.820
C04297=1148.233,348.821,-79.692,-176.466,9.147,148.820
C04298=1148.228,349.068,-79.726,-176.463,9.151,148.820
C04299=1148.225,349.316,-79.761,-176.460,9.155,148.821
C04300=1148.221,349.563,-79.795,-176.458,9.159,148.821
C04301=1148.217,349.811,-79.829,-176.455,9.163,148.821
C04302=1148.213,350.059,-79.864,-176.453,9.166,148.821
C04303=1148.208,350.306,-79.898,-176.450,9.170,148.822
C04304=1148.205,350.554,-79.932,-176.448,9.174,148.822
C04305=1148.200,350.801,-79.967,-176.445,9.178,148.822
C04306=1148.197,351.049,-80.001,-176.442,9.182,148.823
C04307=1148.193,351.296,-80.036,-176.441,9.186,148.823
C04308=1148.189,351.544,-80.071,-176.438,9.190,148.823
C04309=1148.185,351.791,-80.105,-176.435,9.193,148.823
C04310=1148.181,352.039,-80.140,-176.433,9.197,148.824
C04311=1148.177,352.287,-80.174,-176.431,9.201,148.824
C04312=1148.173,352.534,-80.209,-176.428,9.205,148.824
C04313=1148.169,352.782,-80.243,-176.425,9.209,148.825
C04314=1148.165,353.029,-80.279,-176.423,9.212,148.825
C04315=1148.161,353.276,-80.312,-176.420,9.217,148.826
C04316=1148.157,353.525,-80.347,-176.418,9.220,148.826
C04317=1148.153,353.772,-80.382,-176.415,9.224,148.826
C04318=1148.150,354.020,-80.416,-176.413,9.229,148.826
C04319=1148.146,354.267,-80.452,-176.410,9.232,148.827
C04320=1148.141,354.515,-80.486,-176.408,9.236,148.827
C04321=1148.137,354.763,-80.521,-176.405,9.239,148.827
C04322=1148.134,355.009,-80.555,-176.403,9.244,148.828
C04323=1148.130,355.257,-80.590,-176.400,9.248,148.828
C04324=1148.125,355.505,-80.625,-176.398,9.251,148.828
C04325=1148.122,355.752,-80.660,-176.395,9.256,148.829
C04326=1148.118,356.000,-80.695,-176.393,9.259,148.829
C04327=1148.114,356.248,-80.729,-176.390,9.263,148.829
C04328=1148.110,356.495,-80.765,-176.388,9.267,148.830
C04329=1148.106,356.743,-80.799,-176.385,9.271,148.830
C04330=1148.102,356.990,-80.835,-176.383,9.275,148.830
C04331=1148.098,357.238,-80.869,-176.380,9.279,148.831
C04332=1148.094,357.485,-80.904,-176.378,9.283,148.831
C04333=1148.090,357.733,-80.939,-176.375,9.287,148.831
C04334=1148.087,357.980,-80.974,-176.373,9.290,148.831
C04335=1148.082,358.228,-81.009,-176.370,9.294,148.832
C04336=1148.079,358.475,-81.044,-176.367,9.299,148.832
C04337=1148.074,358.723,-81.079,-176.365,9.302,148.833
C04338=1148.070,358.970,-81.114,-176.362,9.306,148.833
C04339=1148.066,359.218,-81.149,-176.360,9.311,148.833
C04340=1148.063,359.465,-81.184,-176.358,9.314,148.834
C04341=1148.059,359.712,-81.219,-176.355,9.318,148.834
C04342=1148.055,359.960,-81.254,-176.352,9.322,148.834
C04343=1148.052,360.208,-81.290,-176.349,9.326,148.835
C04344=1148.047,360.455,-81.324,-176.347,9.330,148.835
C04345=1148.043,360.703,-81.360,-176.344,9.334,148.835
C04346=1148.040,360.950,-81.395,-176.342,9.338,148.835
C04347=1148.035,361.198,-81.430,-176.340,9.342,148.836
C04348=1148.031,361.445,-81.465,-176.337,9.346,148.836
C04349=1148.028,361.693,-81.501,-176.334,9.350,148.837
C04350=1148.024,361.940,-81.536,-176.331,9.354,148.837
C04351=1148.019,362.188,-81.571,-176.329,9.358,148.837
C04352=1148.016,362.435,-81.606,-176.327,9.362,148.838
C04353=1148.012,362.683,-81.642,-176.324,9.366,148.838
C04354=1148.008,362.929,-81.677,-176.321,9.370,148.838
C04355=1148.004,363.177,-81.713,-176.319,9.374,148.838
C04356=1148.000,363.425,-81.748,-176.316,9.378,148.839
C04357=1147.997,363.673,-81.783,-176.313,9.382,148.839
C04358=1147.993,363.920,-81.819,-176.311,9.387,148.840
C04359=1147.989,364.167,-81.854,-176.309,9.390,148.840
C04360=1147.984,364.415,-81.890,-176.306,9.394,148.840
C04361=1147.981,364.662,-81.926,-176.303,9.398,148.841
C04362=1147.976,364.945,-81.966,-176.300,9.404,148.841
C04363=1147.973,365.229,-82.006,-176.297,9.408,148.841
C04364=1147.968,365.512,-82.047,-176.294,9.413,148.842
C04365=1147.964,365.795,-82.088,-176.291,9.417,148.842
C04366=1147.959,366.042,-82.124,-176.289,9.421,148.843
C04367=1147.955,366.290,-82.159,-176.286,9.425,148.843
C04368=1147.951,366.537,-82.195,-176.284,9.429,148.843
C04369=1147.948,366.785,-82.230,-176.281,9.433,148.844
C04370=1147.944,367.032,-82.266,-176.278,9.438,148.844
C04371=1147.940,367.280,-82.302,-176.276,9.442,148.844
C04372=1147.935,367.527,-82.337,-176.273,9.446,148.845
C04373=1147.932,367.775,-82.373,-176.270,9.450,148.845
C04374=1147.928,368.022,-82.408,-176.268,9.454,148.846
C04375=1147.924,368.270,-82.444,-176.266,9.458,148.846
C04376=1147.920,368.517,-82.480,-176.263,9.462,148.846
C04377=1147.917,368.764,-82.516,-176.260,9.467,148.847
C04378=1147.913,369.012,-82.552,-176.257,9.471,148.847
C04379=1147.908,369.259,-82.588,-176.255,9.475,148.847
C04380=1147.904,369.506,-82.623,-176.253,9.479,148.848
C04381=1147.901,369.754,-82.659,-176.250,9.483,148.848
C04382=1147.897,370.001,-82.696,-176.248,9.487,148.849
C04383=1147.893,370.249,-82.731,-176.245,9.491,148.849
C04384=1147.889,370.496,-82.767,-176.242,9.496,148.849
C04385=1147.885,370.744,-82.803,-176.240,9.499,148.850
C04386=1147.881,370.991,-82.839,-176.238,9.504,148.850
C04387=1147.878,371.238,-82.875,-176.235,9.508,148.851
C04388=1147.873,371.486,-82.911,-176.233,9.512,148.851
C04389=1147.870,371.733,-82.947,-176.230,9.516,148.851
C04390=1147.866,371.980,-82.983,-176.228,9.520,148.852
C04391=1147.862,372.228,-83.019,-176.226,9.524,148.852
C04392=1147.859,372.475,-83.055,-176.223,9.529,148.853
C04393=1147.854,372.723,-83.091,-176.221,9.533,148.853
C04394=1147.851,372.970,-83.127,-176.219,9.537,148.854
C04395=1147.847,373.217,-83.163,-176.216,9.541,148.854
C04396=1147.843,373.464,-83.200,-176.214,9.546,148.855
C04397=1147.839,373.712,-83.235,-176.212,9.549,148.855
C04398=1147.835,373.960,-83.272,-176.209,9.553,148.856
C04399=1147.832,374.207,-83.308,-176.207,9.558,148.856
C04400=1147.828,374.454,-83.345,-176.205,9.561,148.856
C04401=1147.824,374.701,-83.380,-176.203,9.566,148.857
C04402=1147.820,374.949,-83.417,-176.200,9.571,148.858
C04403=1147.816,375.196,-83.453,-176.198,9.574,148.858
C04404=1147.812,375.443,-83.490,-176.196,9.579,148.858
C04405=1147.808,375.691,-83.525,-176.194,9.582,148.859
C04406=1147.804,375.938,-83.562,-176.192,9.587,148.860
C04407=1147.801,376.185,-83.597,-176.190,9.590,148.860
C04408=1147.797,376.433,-83.634,-176.188,9.595,148.861
C04409=1147.793,376.680,-83.671,-176.186,9.599,148.861
C04410=1147.789,376.927,-83.707,-176.184,9.603,148.862
C04411=1147.785,377.175,-83.744,-176.182,9.607,148.862
C04412=1147.781,377.421,-83.780,-176.180,9.612,148.863
C04413=1147.777,377.669,-83.816,-176.178,9.615,148.863
C04414=1147.774,377.916,-83.852,-176.177,9.619,148.864
C04415=1147.770,378.163,-83.889,-176.175,9.624,148.865
C04416=1147.765,378.410,-83.926,-176.173,9.627,148.865
C04417=1147.762,378.658,-83.962,-176.171,9.631,148.866
C04418=1147.758,378.906,-83.999,-176.170,9.635,148.866
C04419=1147.754,379.153,-84.036,-176.168,9.640,148.867
C04420=1147.751,379.400,-84.072,-176.166,9.644,148.867
C04421=1147.746,379.648,-84.108,-176.165,9.648,148.868
C04422=1147.743,379.895,-84.144,-176.163,9.652,148.869
C04423=1147.739,380.142,-84.181,-176.162,9.655,148.869
C04424=1147.735,380.389,-84.218,-176.160,9.659,148.870
C04425=1147.732,380.636,-84.254,-176.159,9.663,148.871
C04426=1147.727,380.883,-84.291,-176.157,9.667,148.871
C04427=1147.724,381.132,-84.328,-176.156,9.671,148.872
C04428=1147.720,381.379,-84.364,-176.155,9.674,148.872
C04429=1147.716,381.626,-84.401,-176.154,9.678,148.873
C04430=1147.712,381.873,-84.438,-176.152,9.682,148.874
C04431=1147.708,382.120,-84.474,-176.151,9.686,148.875
C04432=1147.705,382.367,-84.511,-176.150,9.689,148.875
C04433=1147.701,382.614,-84.548,-176.149,9.694,148.876
C04434=1147.697,382.862,-84.585,-176.148,9.697,148.877
C04435=1147.693,383.109,-84.622,-176.147,9.701,148.877
C04436=1147.690,383.356,-84.658,-176.146,9.704,148.878
C04437=1147.685,383.603,-84.695,-176.146,9.707,148.879
C04438=1147.681,383.850,-84.732,-176.145,9.711,148.879
C04439=1147.677,384.098,-84.769,-176.144,9.715,148.880
C04440=1147.675,384.345,-84.805,-176.144,9.718,148.881
C04441=1147.670,384.592,-84.842,-176.143,9.722,148.882
C04442=1147.666,384.840,-84.879,-176.142,9.725,148.882
C04443=1147.662,385.087,-84.916,-176.142,9.728,148.883
C04444=1147.658,385.334,-84.953,-176.142,9.732,148.884
C04445=1147.655,385.582,-84.989,-176.141,9.735,148.885
C04446=1147.651,385.829,-85.026,-176.142,9.738,148.885
C04447=1147.647,386.076,-85.063,-176.141,9.741,148.886
C04448=1147.643,386.323,-85.100,-176.141,9.744,148.887
C04449=1147.639,386.570,-85.137,-176.141,9.747,148.888
C04450=1147.636,386.818,-85.173,-176.141,9.751,148.889
C04451=1147.632,387.065,-85.210,-176.141,9.753,148.889
C04452=1147.628,387.312,-85.247,-176.141,9.757,148.890
C04453=1147.624,387.559,-85.284,-176.141,9.760,148.891
C04454=1147.620,387.807,-85.321,-176.141,9.762,148.892
C04455=1147.617,388.054,-85.357,-176.141,9.765,148.893
C04456=1147.613,388.301,-85.394,-176.141,9.769,148.894
C04457=1147.609,388.549,-85.431,-176.141,9.771,148.894
C04458=1147.605,388.795,-85.469,-176.142,9.774,148.895
C04459=1147.602,389.043,-85.506,-176.142,9.777,148.896
C04460=1147.598,389.290,-85.543,-176.143,9.780,148.897
C04461=1147.594,389.537,-85.579,-176.143,9.782,148.898
C04462=1147.590,389.784,-85.616,-176.143,9.785,148.898
C04463=1147.587,390.032,-85.653,-176.144,9.788,148.899
C04464=1147.583,390.279,-85.690,-176.144,9.791,148.900
C04465=1147.578,390.527,-85.727,-176.145,9.793,148.901
C04466=1147.574,390.813,-85.770,-176.146,9.796,148.902
C04467=1147.570,391.100,-85.812,-176.146,9.798,148.903
C04468=1147.565,391.386,-85.856,-176.147,9.802,148.904
C04469=1147.561,391.673,-85.899,-176.148,9.805,148.905
C04470=1147.557,391.921,-85.935,-176.148,9.807,148.906
C04471=1147.554,392.168,-85.972,-176.149,9.809,148.906
C04472=1147.550,392.415,-86.009,-176.150,9.812,148.907
C04473=1147.547,392.662,-86.046,-176.151,9.814,148.908
C04474=1147.542,392.909,-86.083,-176.151,9.817,148.909
C04475=1147.538,393.156,-86.120,-176.152,9.819,148.910
C04476=1147.534,393.404,-86.157,-176.153,9.822,148.911
C04477=1147.531,393.651,-86.194,-176.154,9.824,148.911
C04478=1147.527,393.899,-86.231,-176.155,9.826,148.912
C04479=1147.523,394.146,-86.267,-176.156,9.829,148.913
C04480=1147.520,394.392,-86.305,-176.157,9.831,148.914
C04481=1147.515,394.639,-86.342,-176.158,9.833,148.915
C04482=1147.512,394.887,-86.379,-176.159,9.835,148.916
C04483=1147.508,395.134,-86.416,-176.159,9.838,148.917
C04484=1147.504,395.382,-86.453,-176.160,9.840,148.917
C04485=1147.500,395.629,-86.490,-176.162,9.842,148.918
C04486=1147.496,395.876,-86.528,-176.163,9.844,148.919
C04487=1147.493,396.123,-86.564,-176.164,9.846,148.920
C04488=1147.489,396.370,-86.601,-176.165,9.848,148.921
C04489=1147.485,396.617,-86.638,-176.165,9.851,148.922
C04490=1147.481,396.865,-86.675,-176.167,9.853,148.922
C04491=1147.477,397.112,-86.712,-176.167,9.855,148.923
C04492=1147.474,397.359,-86.749,-176.168,9.857,148.924
C04493=1147.469,397.606,-86.786,-176.169,9.859,148.925
C04494=1147.466,397.854,-86.823,-176.171,9.861,148.926
C04495=1147.462,398.101,-86.860,-176.172,9.863,148.926
C04496=1147.459,398.348,-86.896,-176.173,9.865,148.927
C04497=1147.454,398.595,-86.933,-176.174,9.867,148.928
C04498=1147.451,398.843,-86.971,-176.175,9.869,148.929
C04499=1147.447,399.090,-87.008,-176.176,9.871,148.930
C04500=1147.443,399.337,-87.045,-176.177,9.873,148.931
C04501=1147.439,399.584,-87.082,-176.178,9.876,148.931
C04502=1147.435,399.832,-87.119,-176.179,9.878,148.932
C04503=1147.432,400.079,-87.157,-176.180,9.880,148.933
C04504=1147.428,400.325,-87.193,-176.182,9.881,148.934
C04505=1147.424,400.573,-87.230,-176.183,9.883,148.935
C04506=1147.420,400.820,-87.267,-176.184,9.885,148.935
C04507=1147.417,401.068,-87.304,-176.185,9.887,148.936
C04508=1147.413,401.315,-87.341,-176.186,9.889,148.937
C04509=1147.409,401.561,-87.378,-176.187,9.891,148.938
C04510=1147.405,401.809,-87.415,-176.188,9.893,148.939
C04511=1147.401,402.057,-87.452,-176.189,9.895,148.940
C04512=1147.397,402.304,-87.489,-176.190,9.897,148.940
C04513=1147.394,402.551,-87.525,-176.191,9.899,148.941
C04514=1147.390,402.798,-87.562,-176.193,9.900,148.942
C04515=1147.386,403.045,-87.600,-176.194,9.902,148.943
C04516=1147.382,403.292,-87.637,-176.195,9.904,148.944
C04517=1147.378,403.539,-87.674,-176.196,9.906,148.944
C04518=1147.374,403.787,-87.711,-176.197,9.908,148.945
C04519=1147.371,404.035,-87.748,-176.198,9.910,148.946
C04520=1147.367,404.282,-87.785,-176.199,9.912,148.947
C04521=1147.363,404.528,-87.822,-176.200,9.914,148.947
C04522=1147.359,404.775,-87.859,-176.201,9.915,148.948
C04523=1147.356,405.023,-87.896,-176.202,9.917,148.949
C04524=1147.352,405.270,-87.933,-176.204,9.919,148.950
C04525=1147.348,405.517,-87.970,-176.204,9.921,148.950
C04526=1147.344,405.764,-88.007,-176.205,9.923,148.951
C04527=1147.340,406.012,-88.044,-176.206,9.925,148.952
C04528=1147.336,406.259,-88.081,-176.207,9.927,148.953
C04529=1147.332,406.506,-88.118,-176.208,9.929,148.954
C04530=1147.328,406.754,-88.155,-176.209,9.931,148.954
C04531=1147.325,407.001,-88.192,-176.210,9.933,148.955
C04532=1147.322,407.248,-88.229,-176.212,9.934,148.956
C04533=1147.318,407.495,-88.266,-176.212,9.936,148.956
C04534=1147.313,407.742,-88.303,-176.213,9.938,148.957
C04535=1147.310,407.990,-88.340,-176.215,9.940,148.958
C04536=1147.306,408.237,-88.377,-176.215,9.942,148.959
C04537=1147.302,408.484,-88.415,-176.216,9.944,148.960
C04538=1147.298,408.731,-88.451,-176.217,9.946,148.960
C04539=1147.295,408.978,-88.488,-176.218,9.948,148.961
C04540=1147.291,409.226,-88.525,-176.219,9.949,148.962
C04541=1147.287,409.473,-88.562,-176.220,9.951,148.963
C04542=1147.283,409.720,-88.599,-176.220,9.953,148.963
C04543=1147.280,409.967,-88.637,-176.222,9.955,148.964
C04544=1147.276,410.215,-88.673,-176.222,9.957,148.965
C04545=1147.272,410.462,-88.710,-176.223,9.959,148.965
C04546=1147.267,410.709,-88.747,-176.224,9.961,148.966
C04547=1147.264,410.957,-88.784,-176.225,9.963,148.967
C04548=1147.260,411.203,-88.822,-176.226,9.965,148.968
C04549=1147.257,411.450,-88.858,-176.227,9.967,148.968
C04550=1147.253,411.697,-88.895,-176.228,9.968,148.969
C04551=1147.249,411.945,-88.932,-176.228,9.970,148.970
C04552=1147.245,412.193,-88.969,-176.229,9.972,148.971
C04553=1147.241,412.440,-89.006,-176.229,9.975,148.971
C04554=1147.237,412.686,-89.044,-176.230,9.977,148.972
C04555=1147.233,412.933,-89.080,-176.231,9.979,148.973
C04556=1147.230,413.181,-89.118,-176.232,9.980,148.973
C04557=1147.226,413.429,-89.155,-176.233,9.982,148.974
C04558=1147.221,413.676,-89.191,-176.234,9.984,148.975
C04559=1147.218,413.922,-89.228,-176.234,9.986,148.975
C04560=1147.215,414.170,-89.266,-176.235,9.988,148.976
C04561=1147.211,414.417,-89.302,-176.235,9.991,148.977
C04562=1147.207,414.664,-89.339,-176.236,9.992,148.978
C04563=1147.204,414.912,-89.377,-176.237,9.994,148.978
C04564=1147.201,415.159,-89.414,-176.238,9.996,148.979
C04565=1147.199,415.406,-89.451,-176.238,9.998,148.980
C04566=1147.198,415.706,-89.495,-176.239,10.001,148.981
C04567=1147.198,416.007,-89.540,-176.240,10.003,148.981
C04568=1147.199,416.307,-89.584,-176.241,10.005,148.982
C04569=1147.201,416.607,-89.629,-176.241,10.007,148.983
C04570=1147.204,416.940,-89.677,-176.242,10.009,148.984
C04571=1147.209,417.272,-89.726,-176.243,10.012,148.985
C04572=1146.788,417.275,-89.775,-176.245,10.023,148.988
C04573=1146.785,417.040,-89.741,-176.245,10.021,148.987
C04574=1146.782,416.805,-89.707,-176.244,10.020,148.987
C04575=1146.780,416.570,-89.672,-176.244,10.018,148.986
C04576=1146.778,416.335,-89.638,-176.243,10.016,148.986
C04577=1146.777,416.100,-89.602,-176.242,10.015,148.985
C04578=1146.777,415.865,-89.568,-176.242,10.013,148.984
C04579=1146.778,415.629,-89.533,-176.241,10.011,148.984
C04580=1146.778,415.394,-89.497,-176.240,10.009,148.983
C04581=1146.781,415.147,-89.461,-176.240,10.006,148.982
C04582=1146.783,414.900,-89.424,-176.239,10.005,148.982
C04583=1146.786,414.653,-89.387,-176.239,10.003,148.981
C04584=1146.790,414.405,-89.350,-176.238,10.001,148.980
C04585=1146.794,414.158,-89.313,-176.237,9.999,148.980
C04586=1146.798,413.912,-89.276,-176.236,9.997,148.979
C04587=1146.801,413.664,-89.239,-176.236,9.995,148.978
C04588=1146.805,413.417,-89.202,-176.235,9.993,148.977
C04589=1146.809,413.169,-89.165,-176.234,9.991,148.977
C04590=1146.813,412.922,-89.128,-176.233,9.989,148.976
C04591=1146.817,412.675,-89.090,-176.233,9.987,148.975
C04592=1146.821,412.428,-89.053,-176.232,9.985,148.975
C04593=1146.825,412.181,-89.016,-176.231,9.983,148.974
C04594=1146.828,411.934,-88.980,-176.230,9.982,148.973
C04595=1146.831,411.686,-88.942,-176.229,9.980,148.972
C04596=1146.835,411.439,-88.905,-176.228,9.978,148.972
C04597=1146.840,411.192,-88.869,-176.227,9.976,148.971
C04598=1146.844,410.945,-88.832,-176.227,9.973,148.970
C04599=1146.847,410.697,-88.794,-176.226,9.971,148.969
C04600=1146.851,410.450,-88.757,-176.226,9.969,148.969
C04601=1146.855,410.203,-88.720,-176.224,9.967,148.968
C04602=1146.859,409.956,-88.683,-176.224,9.966,148.967
C04603=1146.863,409.708,-88.646,-176.223,9.964,148.966
C04604=1146.866,409.461,-88.610,-176.222,9.962,148.966
C04605=1146.870,409.214,-88.573,-176.221,9.960,148.965
C04606=1146.874,408.967,-88.535,-176.220,9.958,148.964
C04607=1146.877,408.720,-88.498,-176.219,9.956,148.964
C04608=1146.881,408.472,-88.461,-176.218,9.954,148.963
C04609=1146.886,408.225,-88.424,-176.217,9.953,148.962
C04610=1146.890,407.978,-88.387,-176.216,9.951,148.961
C04611=1146.893,407.731,-88.349,-176.215,9.949,148.961
C04612=1146.897,407.484,-88.313,-176.214,9.947,148.960
C04613=1146.901,407.236,-88.276,-176.213,9.945,148.959
C04614=1146.904,406.989,-88.240,-176.212,9.943,148.958
C04615=1146.908,406.742,-88.202,-176.211,9.941,148.957
C04616=1146.912,406.495,-88.165,-176.210,9.939,148.957
C04617=1146.916,406.248,-88.128,-176.209,9.937,148.956
C04618=1146.920,406.001,-88.091,-176.208,9.935,148.955
C04619=1146.923,405.753,-88.054,-176.208,9.933,148.955
C04620=1146.927,405.506,-88.017,-176.206,9.931,148.954
C04621=1146.931,405.259,-87.979,-176.205,9.930,148.953
C04622=1146.935,405.012,-87.942,-176.204,9.928,148.952
C04623=1146.938,404.764,-87.906,-176.203,9.926,148.951
C04624=1146.942,404.517,-87.869,-176.202,9.924,148.951
C04625=1146.946,404.270,-87.832,-176.201,9.922,148.950
C04626=1146.950,404.023,-87.795,-176.200,9.920,148.949
C04627=1146.954,403.775,-87.757,-176.199,9.918,148.948
C04628=1146.958,403.528,-87.720,-176.198,9.916,148.947
C04629=1146.962,403.281,-87.684,-176.196,9.915,148.947
C04630=1146.966,403.034,-87.647,-176.195,9.913,148.946
C04631=1146.969,402.786,-87.610,-176.194,9.911,148.945
C04632=1146.973,402.539,-87.572,-176.193,9.909,148.944
C04633=1146.976,402.292,-87.536,-176.192,9.907,148.944
C04634=1146.981,402.045,-87.499,-176.191,9.905,148.943
C04635=1146.984,401.797,-87.462,-176.190,9.903,148.942
C04636=1146.988,401.550,-87.425,-176.189,9.901,148.941
C04637=1146.992,401.304,-87.387,-176.187,9.900,148.940
C04638=1146.996,401.056,-87.350,-176.186,9.898,148.939
C04639=1147.000,400.809,-87.313,-176.185,9.896,148.939
C04640=1147.004,400.561,-87.276,-176.184,9.894,148.938
C04641=1147.008,400.314,-87.239,-176.183,9.892,148.937
C04642=1147.011,400.068,-87.202,-176.182,9.890,148.936
C04643=1147.014,399.820,-87.165,-176.181,9.888,148.935
C04644=1147.018,399.573,-87.128,-176.180,9.886,148.935
C04645=1147.022,399.326,-87.091,-176.179,9.884,148.934
C04646=1147.027,399.078,-87.055,-176.178,9.881,148.933
C04647=1147.030,398.831,-87.017,-176.177,9.879,148.932
C04648=1147.034,398.584,-86.980,-176.176,9.877,148.931
C04649=1147.038,398.337,-86.943,-176.175,9.875,148.930
C04650=1147.042,398.090,-86.906,-176.173,9.873,148.930
C04651=1147.045,397.842,-86.869,-176.172,9.871,148.929
C04652=1147.049,397.595,-86.833,-176.171,9.869,148.928
C04653=1147.053,397.348,-86.795,-176.170,9.867,148.927
C04654=1147.057,397.101,-86.758,-176.169,9.865,148.926
C04655=1147.060,396.853,-86.721,-176.168,9.863,148.926
C04656=1147.064,396.606,-86.684,-176.167,9.861,148.925
C04657=1147.068,396.359,-86.647,-176.166,9.859,148.924
C04658=1147.072,396.112,-86.610,-176.165,9.857,148.923
C04659=1147.076,395.864,-86.572,-176.164,9.855,148.922
C04660=1147.080,395.617,-86.536,-176.163,9.853,148.921
C04661=1147.083,395.370,-86.499,-176.162,9.851,148.921
C04662=1147.087,395.123,-86.462,-176.161,9.848,148.920
C04663=1147.091,394.875,-86.425,-176.160,9.846,148.919
C04664=1147.095,394.629,-86.388,-176.159,9.844,148.918
C04665=1147.099,394.381,-86.351,-176.158,9.842,148.917
C04666=1147.103,394.134,-86.314,-176.157,9.839,148.916
C04667=1147.106,393.886,-86.277,-176.156,9.837,148.915
C04668=1147.110,393.639,-86.240,-176.155,9.835,148.915
C04669=1147.114,393.392,-86.203,-176.155,9.832,148.914
C04670=1147.117,393.146,-86.166,-176.154,9.830,148.913
C04671=1147.121,392.898,-86.129,-176.152,9.828,148.912
C04672=1147.125,392.651,-86.092,-176.152,9.825,148.911
C04673=1147.129,392.403,-86.055,-176.151,9.823,148.910
C04674=1147.133,392.156,-86.018,-176.151,9.820,148.910
C04675=1147.137,391.908,-85.981,-176.150,9.818,148.909
C04676=1147.141,391.662,-85.943,-176.149,9.815,148.908
C04677=1147.145,391.375,-85.901,-176.149,9.813,148.907
C04678=1147.149,391.088,-85.859,-176.148,9.809,148.906
C04679=1147.153,390.802,-85.816,-176.147,9.806,148.905
C04680=1147.159,390.515,-85.773,-176.147,9.804,148.904
C04681=1147.162,390.267,-85.735,-176.146,9.801,148.903
C04682=1147.165,390.020,-85.699,-176.145,9.799,148.902
C04683=1147.169,389.774,-85.662,-176.144,9.796,148.901
C04684=1147.173,389.526,-85.625,-176.144,9.793,148.901
C04685=1147.177,389.279,-85.588,-176.144,9.790,148.900
C04686=1147.181,389.031,-85.551,-176.143,9.788,148.899
C04687=1147.185,388.784,-85.514,-176.143,9.785,148.898
C04688=1147.188,388.537,-85.478,-176.143,9.782,148.897
C04689=1147.192,388.289,-85.440,-176.143,9.780,148.897
C04690=1147.196,388.042,-85.403,-176.143,9.776,148.896
C04691=1147.200,387.796,-85.366,-176.143,9.773,148.895
C04692=1147.204,387.548,-85.329,-176.142,9.770,148.894
C04693=1147.207,387.301,-85.292,-176.142,9.768,148.893
C04694=1147.211,387.054,-85.256,-176.142,9.764,148.892
C04695=1147.215,386.806,-85.219,-176.142,9.762,148.892
C04696=1147.219,386.559,-85.182,-176.142,9.758,148.891
C04697=1147.223,386.312,-85.145,-176.142,9.756,148.890
C04698=1147.226,386.064,-85.108,-176.142,9.752,148.889
C04699=1147.230,385.817,-85.071,-176.143,9.749,148.889
C04700=1147.234,385.570,-85.035,-176.143,9.746,148.888
C04701=1147.238,385.323,-84.998,-176.143,9.743,148.887
C04702=1147.242,385.076,-84.961,-176.144,9.739,148.886
C04703=1147.246,384.828,-84.924,-176.144,9.736,148.886
C04704=1147.249,384.581,-84.887,-176.145,9.732,148.885
C04705=1147.253,384.334,-84.851,-176.145,9.729,148.884
C04706=1147.257,384.087,-84.814,-176.146,9.726,148.883
C04707=1147.261,383.839,-84.777,-176.146,9.722,148.883
C04708=1147.265,383.592,-84.740,-176.148,9.718,148.882
C04709=1147.268,383.345,-84.703,-176.148,9.715,148.881
C04710=1147.272,383.097,-84.667,-176.149,9.712,148.881
C04711=1147.276,382.850,-84.630,-176.150,9.708,148.880
C04712=1147.280,382.603,-84.593,-176.150,9.704,148.879
C04713=1147.284,382.356,-84.557,-176.152,9.701,148.879
C04714=1147.287,382.108,-84.519,-176.152,9.697,148.878
C04715=1147.291,381.861,-84.482,-176.154,9.693,148.877
C04716=1147.295,381.614,-84.446,-176.155,9.689,148.876
C04717=1147.299,381.367,-84.409,-176.156,9.686,148.876
C04718=1147.303,381.120,-84.372,-176.157,9.682,148.875
C04719=1147.307,380.873,-84.336,-176.159,9.678,148.875
C04720=1147.310,380.626,-84.299,-176.160,9.674,148.874
C04721=1147.314,380.377,-84.263,-176.161,9.670,148.873
C04722=1147.318,380.130,-84.226,-176.163,9.666,148.873
C04723=1147.322,379.883,-84.190,-176.164,9.662,148.872
C04724=1147.326,379.636,-84.153,-176.166,9.659,148.871
C04725=1147.330,379.389,-84.116,-176.167,9.655,148.871
C04726=1147.333,379.141,-84.080,-176.169,9.651,148.870
C04727=1147.337,378.894,-84.044,-176.171,9.646,148.870
C04728=1147.342,378.647,-84.007,-176.173,9.642,148.869
C04729=1147.345,378.400,-83.970,-176.174,9.639,148.868
C04730=1147.348,378.152,-83.933,-176.176,9.635,148.868
C04731=1147.353,377.904,-83.897,-176.178,9.630,148.867
C04732=1147.356,377.657,-83.861,-176.180,9.626,148.867
C04733=1147.360,377.410,-83.824,-176.182,9.623,148.866
C04734=1147.364,377.163,-83.788,-176.184,9.618,148.866
C04735=1147.368,376.916,-83.752,-176.186,9.615,148.865
C04736=1147.371,376.669,-83.715,-176.188,9.610,148.864
C04737=1147.376,376.421,-83.679,-176.190,9.606,148.864
C04738=1147.380,376.174,-83.642,-176.192,9.602,148.863
C04739=1147.383,375.927,-83.606,-176.194,9.598,148.863
C04740=1147.388,375.679,-83.570,-176.196,9.594,148.862
C04741=1147.391,375.432,-83.534,-176.198,9.590,148.862
C04742=1147.395,375.184,-83.497,-176.200,9.585,148.861
C04743=1147.399,374.937,-83.461,-176.202,9.582,148.861
C04744=1147.403,374.690,-83.424,-176.205,9.577,148.861
C04745=1147.407,374.443,-83.389,-176.207,9.573,148.860
C04746=1147.411,374.196,-83.352,-176.209,9.569,148.860
C04747=1147.414,373.948,-83.316,-176.211,9.565,148.859
C04748=1147.418,373.701,-83.280,-176.214,9.560,148.858
C04749=1147.422,373.453,-83.244,-176.215,9.557,148.858
C04750=1147.426,373.206,-83.207,-176.218,9.552,148.858
C04751=1147.430,372.959,-83.172,-176.220,9.548,148.857
C04752=1147.433,372.711,-83.136,-176.223,9.544,148.857
C04753=1147.438,372.464,-83.099,-176.225,9.540,148.856
C04754=1147.441,372.216,-83.064,-176.228,9.536,148.856
C04755=1147.445,371.969,-83.027,-176.230,9.531,148.855
C04756=1147.449,371.722,-82.991,-176.233,9.527,148.855
C04757=1147.453,371.474,-82.956,-176.235,9.523,148.855
C04758=1147.457,371.227,-82.919,-176.237,9.519,148.854
C04759=1147.460,370.980,-82.883,-176.240,9.515,148.854
C04760=1147.465,370.732,-82.847,-176.243,9.511,148.853
C04761=1147.468,370.485,-82.811,-176.245,9.506,148.853
C04762=1147.472,370.237,-82.775,-176.248,9.502,148.852
C04763=1147.476,369.990,-82.739,-176.250,9.499,148.852
C04764=1147.480,369.743,-82.703,-176.252,9.494,148.852
C04765=1147.483,369.495,-82.667,-176.255,9.490,148.851
C04766=1147.488,369.247,-82.631,-176.258,9.486,148.851
C04767=1147.492,369.001,-82.596,-176.260,9.481,148.851
C04768=1147.496,368.753,-82.561,-176.263,9.477,148.850
C04769=1147.499,368.506,-82.524,-176.265,9.474,148.850
C04770=1147.503,368.258,-82.488,-176.268,9.469,148.849
C04771=1147.507,368.011,-82.453,-176.270,9.465,148.849
C04772=1147.511,367.763,-82.417,-176.273,9.461,148.849
C04773=1147.514,367.516,-82.381,-176.275,9.456,148.848
C04774=1147.519,367.268,-82.345,-176.278,9.452,148.848
C04775=1147.523,367.021,-82.310,-176.280,9.449,148.848
C04776=1147.527,366.774,-82.275,-176.283,9.445,148.847
C04777=1147.530,366.526,-82.239,-176.286,9.440,148.847
C04778=1147.535,366.278,-82.203,-176.289,9.436,148.847
C04779=1147.538,366.031,-82.167,-176.291,9.432,148.846
C04780=1147.542,365.783,-82.132,-176.294,9.428,148.846
C04781=1147.547,365.501,-82.091,-176.296,9.423,148.845
C04782=1147.551,365.217,-82.051,-176.300,9.418,148.845
C04783=1147.556,364.934,-82.010,-176.302,9.414,148.845
C04784=1147.560,364.651,-81.969,-176.306,9.409,148.844
C04785=1147.564,364.403,-81.934,-176.308,9.406,148.844
C04786=1147.568,364.156,-81.898,-176.311,9.401,148.844
C04787=1147.571,363.908,-81.862,-176.313,9.397,148.843
C04788=1147.576,363.661,-81.827,-176.316,9.393,148.843
C04789=1147.579,363.414,-81.792,-176.319,9.389,148.842
C04790=1147.583,363.166,-81.756,-176.321,9.385,148.842
C04791=1147.587,362.918,-81.721,-176.324,9.381,148.842
C04792=1147.590,362.671,-81.686,-176.326,9.377,148.841
C04793=1147.595,362.424,-81.651,-176.329,9.372,148.841
C04794=1147.598,362.176,-81.615,-176.331,9.369,148.841
C04795=1147.602,361.929,-81.579,-176.334,9.365,148.840
C04796=1147.607,361.682,-81.545,-176.337,9.361,148.840
C04797=1147.610,361.434,-81.509,-176.340,9.357,148.840
C04798=1147.614,361.187,-81.474,-176.341,9.353,148.839
C04799=1147.618,360.938,-81.439,-176.344,9.349,148.839
C04800=1147.622,360.692,-81.404,-176.347,9.345,148.839
C04801=1147.626,360.444,-81.368,-176.350,9.340,148.838
C04802=1147.630,360.197,-81.333,-176.352,9.337,148.838
C04803=1147.634,359.949,-81.298,-176.355,9.333,148.838
C04804=1147.638,359.702,-81.263,-176.358,9.329,148.837
C04805=1147.642,359.454,-81.228,-176.359,9.325,148.837
C04806=1147.645,359.206,-81.192,-176.362,9.321,148.837
C04807=1147.650,358.959,-81.157,-176.365,9.317,148.836
C04808=1147.654,358.711,-81.122,-176.367,9.313,148.836
C04809=1147.657,358.464,-81.087,-176.370,9.309,148.836
C04810=1147.662,358.216,-81.052,-176.373,9.305,148.835
C04811=1147.665,357.969,-81.017,-176.375,9.302,148.835
C04812=1147.669,357.722,-80.983,-176.377,9.297,148.835
C04813=1147.673,357.474,-80.947,-176.380,9.293,148.834
C04814=1147.677,357.226,-80.913,-176.382,9.290,148.834
C04815=1147.681,356.979,-80.877,-176.385,9.285,148.834
C04816=1147.685,356.731,-80.843,-176.388,9.281,148.833
C04817=1147.689,356.484,-80.807,-176.390,9.278,148.833
C04818=1147.693,356.236,-80.773,-176.393,9.274,148.833
C04819=1147.697,355.988,-80.738,-176.395,9.270,148.832
C04820=1147.701,355.742,-80.703,-176.398,9.266,148.832
C04821=1147.705,355.493,-80.668,-176.400,9.262,148.832
C04822=1147.709,355.246,-80.633,-176.402,9.258,148.831
C04823=1147.712,354.999,-80.599,-176.405,9.254,148.831
C04824=1147.716,354.751,-80.564,-176.407,9.251,148.831
C04825=1147.721,354.504,-80.529,-176.410,9.247,148.830
C04826=1147.725,354.256,-80.494,-176.413,9.242,148.830
C04827=1147.728,354.009,-80.460,-176.415,9.239,148.830
C04828=1147.732,353.761,-80.425,-176.418,9.235,148.830
C04829=1147.737,353.514,-80.390,-176.420,9.231,148.829
C04830=1147.740,353.266,-80.356,-176.423,9.227,148.829
C04831=1147.744,353.018,-80.321,-176.425,9.223,148.828
C04832=1147.748,352.770,-80.287,-176.428,9.220,148.828
C04833=1147.751,352.523,-80.252,-176.430,9.215,148.828
C04834=1147.756,352.276,-80.217,-176.433,9.211,148.828
C04835=1147.760,352.028,-80.182,-176.435,9.208,148.827
C04836=1147.764,351.781,-80.148,-176.438,9.203,148.827
C04837=1147.768,351.532,-80.114,-176.440,9.200,148.827
C04838=1147.772,351.285,-80.079,-176.443,9.196,148.826
C04839=1147.776,351.037,-80.045,-176.445,9.192,148.826
C04840=1147.780,350.790,-80.010,-176.448,9.188,148.826
C04841=1147.784,350.542,-79.975,-176.451,9.184,148.825
C04842=1147.788,350.295,-79.941,-176.453,9.181,148.825
C04843=1147.792,350.048,-79.907,-176.456,9.177,148.825
C04844=1147.795,349.800,-79.872,-176.458,9.173,148.825
C04845=1147.800,349.553,-79.838,-176.460,9.169,148.824
C04846=1147.804,349.304,-79.803,-176.463,9.165,148.824
C04847=1147.808,349.057,-79.769,-176.466,9.162,148.824
C04848=1147.812,348.809,-79.734,-176.468,9.157,148.823
C04849=1147.816,348.562,-79.700,-176.470,9.154,148.823
C04850=1147.820,348.314,-79.666,-176.473,9.150,148.823
C04851=1147.824,348.066,-79.632,-176.475,9.146,148.822
C04852=1147.828,347.819,-79.598,-176.478,9.142,148.822
C04853=1147.831,347.571,-79.564,-176.480,9.139,148.822
C04854=1147.836,347.324,-79.529,-176.483,9.135,148.821
C04855=1147.839,347.076,-79.495,-176.486,9.130,148.821
C04856=1147.844,346.828,-79.461,-176.488,9.127,148.821
C04857=1147.848,346.581,-79.427,-176.491,9.123,148.821
C04858=1147.852,346.333,-79.392,-176.493,9.120,148.820
C04859=1147.856,346.085,-79.359,-176.496,9.115,148.820
C04860=1147.860,345.838,-79.324,-176.498,9.112,148.820
C04861=1147.864,345.590,-79.290,-176.501,9.108,148.819
C04862=1147.868,345.343,-79.256,-176.503,9.105,148.819
C04863=1147.872,345.095,-79.222,-176.506,9.100,148.819
C04864=1147.876,344.847,-79.188,-176.508,9.096,148.819
C04865=1147.880,344.600,-79.154,-176.511,9.093,148.818
C04866=1147.884,344.353,-79.120,-176.514,9.089,148.818
C04867=1147.888,344.104,-79.086,-176.516,9.085,148.818
C04868=1147.892,343.857,-79.052,-176.518,9.081,148.817
C04869=1147.896,343.610,-79.018,-176.521,9.078,148.817
C04870=1147.900,343.361,-78.984,-176.524,9.074,148.817
C04871=1147.904,343.114,-78.950,-176.526,9.070,148.817
C04872=1147.908,342.867,-78.916,-176.529,9.066,148.816
C04873=1147.912,342.618,-78.882,-176.531,9.063,148.816
C04874=1147.916,342.371,-78.848,-176.534,9.059,148.816
C04875=1147.920,342.123,-78.815,-176.536,9.055,148.816
C04876=1147.925,341.876,-78.781,-176.539,9.051,148.815
C04877=1147.928,341.627,-78.747,-176.541,9.048,148.815
C04878=1147.932,341.380,-78.713,-176.544,9.044,148.815
C04879=1147.936,341.133,-78.680,-176.546,9.040,148.815
C04880=1147.941,340.885,-78.646,-176.549,9.036,148.814
C04881=1147.944,340.637,-78.612,-176.552,9.032,148.814
C04882=1147.948,340.390,-78.578,-176.554,9.029,148.814
C04883=1147.953,340.141,-78.544,-176.557,9.024,148.813
C04884=1147.957,339.894,-78.511,-176.559,9.021,148.813
C04885=1147.961,339.614,-78.473,-176.562,9.017,148.813
C04886=1147.965,339.333,-78.434,-176.564,9.013,148.813
C04887=1147.970,339.054,-78.397,-176.567,9.009,148.812
C04888=1147.975,338.773,-78.358,-176.570,9.005,148.812
C04889=1147.979,338.526,-78.325,-176.573,9.000,148.812
C04890=1147.983,338.277,-78.291,-176.575,8.997,148.811
C04891=1147.986,338.030,-78.258,-176.578,8.993,148.811
C04892=1147.990,337.782,-78.224,-176.580,8.990,148.811
C04893=1147.995,337.534,-78.191,-176.583,8.985,148.811
C04894=1147.999,337.287,-78.157,-176.586,8.982,148.810
C04895=1148.003,337.039,-78.123,-176.588,8.978,148.810
C04896=1148.007,336.791,-78.090,-176.590,8.975,148.810
C04897=1148.011,336.543,-78.057,-176.593,8.970,148.810
C04898=1148.015,336.296,-78.023,-176.596,8.967,148.809
C04899=1148.019,336.048,-77.990,-176.599,8.963,148.809
C04900=1148.023,335.801,-77.957,-176.601,8.960,148.809
C04901=1148.027,335.552,-77.923,-176.604,8.956,148.809
C04902=1148.031,335.305,-77.890,-176.606,8.952,148.808
C04903=1148.035,335.057,-77.856,-176.609,8.948,148.808
C04904=1148.039,334.810,-77.823,-176.611,8.945,148.808
C04905=1148.044,334.562,-77.789,-176.614,8.941,148.808
C04906=1148.048,334.314,-77.756,-176.616,8.937,148.807
C04907=1148.052,334.066,-77.723,-176.619,8.933,148.807
C04908=1148.056,333.818,-77.690,-176.621,8.930,148.807
C04909=1148.060,333.571,-77.657,-176.624,8.926,148.807
C04910=1148.063,333.323,-77.624,-176.627,8.923,148.807
C04911=1148.067,333.075,-77.591,-176.629,8.919,148.806
C04912=1148.071,332.827,-77.557,-176.631,8.915,148.806
C04913=1148.075,332.579,-77.524,-176.634,8.912,148.806
C04914=1148.080,332.332,-77.491,-176.637,8.908,148.805
C04915=1148.084,332.084,-77.458,-176.639,8.904,148.805
C04916=1148.088,331.836,-77.425,-176.642,8.900,148.805
C04917=1148.092,331.589,-77.392,-176.644,8.897,148.805
C04918=1148.096,331.341,-77.358,-176.647,8.893,148.805
C04919=1148.100,331.093,-77.325,-176.649,8.890,148.804
C04920=1148.104,330.845,-77.292,-176.652,8.886,148.804
C04921=1148.108,330.598,-77.259,-176.655,8.882,148.804
C04922=1148.113,330.350,-77.226,-176.657,8.879,148.804
C04923=1148.116,330.102,-77.193,-176.659,8.875,148.803
C04924=1148.120,329.854,-77.161,-176.662,8.871,148.803
C04925=1148.125,329.606,-77.128,-176.665,8.867,148.803
C04926=1148.129,329.359,-77.095,-176.667,8.864,148.803
C04927=1148.133,329.111,-77.061,-176.670,8.860,148.802
C04928=1148.137,328.863,-77.028,-176.672,8.857,148.802
C04929=1148.140,328.616,-76.996,-176.675,8.853,148.802
C04930=1148.145,328.367,-76.963,-176.678,8.849,148.802
C04931=1148.149,328.120,-76.930,-176.680,8.846,148.802
C04932=1148.153,327.872,-76.897,-176.683,8.842,148.801
C04933=1148.157,327.624,-76.864,-176.685,8.839,148.801
C04934=1148.161,327.376,-76.832,-176.688,8.835,148.801
C04935=1148.165,327.128,-76.799,-176.690,8.831,148.801
C04936=1148.169,326.881,-76.766,-176.693,8.828,148.801
C04937=1148.174,326.632,-76.733,-176.696,8.824,148.800
C04938=1148.177,326.385,-76.701,-176.698,8.821,148.800
C04939=1148.181,326.137,-76.667,-176.701,8.817,148.800
C04940=1148.186,325.889,-76.635,-176.703,8.813,148.800
C04941=1148.189,325.641,-76.602,-176.706,8.809,148.799
C04942=1148.194,325.393,-76.570,-176.708,8.806,148.799
C04943=1148.198,325.146,-76.537,-176.711,8.803,148.799
C04944=1148.202,324.898,-76.504,-176.714,8.799,148.799
C04945=1148.206,324.650,-76.472,-176.716,8.795,148.799
C04946=1148.210,324.403,-76.439,-176.719,8.791,148.798
C04947=1148.215,324.154,-76.407,-176.721,8.788,148.798
C04948=1148.218,323.907,-76.374,-176.723,8.785,148.798
C04949=1148.223,323.658,-76.342,-176.726,8.781,148.798
C04950=1148.226,323.411,-76.309,-176.729,8.777,148.798
C04951=1148.230,323.163,-76.277,-176.732,8.773,148.797
C04952=1148.235,322.915,-76.243,-176.734,8.770,148.797
C04953=1148.239,322.668,-76.212,-176.736,8.767,148.797
C04954=1148.243,322.419,-76.180,-176.740,8.763,148.797
C04955=1148.247,322.172,-76.147,-176.742,8.760,148.797
C04956=1148.251,321.924,-76.115,-176.745,8.756,148.797
C04957=1148.255,321.676,-76.082,-176.747,8.752,148.796
C04958=1148.259,321.428,-76.050,-176.749,8.749,148.796
C04959=1148.263,321.180,-76.018,-176.752,8.745,148.796
C04960=1148.267,320.933,-75.985,-176.755,8.742,148.796
C04961=1148.271,320.685,-75.953,-176.757,8.739,148.796
C04962=1148.276,320.436,-75.921,-176.760,8.734,148.795
C04963=1148.279,320.189,-75.888,-176.762,8.731,148.795
C04964=1148.283,319.941,-75.856,-176.765,8.727,148.795
C04965=1148.288,319.693,-75.824,-176.768,8.724,148.795
C04966=1148.292,319.445,-75.792,-176.770,8.721,148.795
C04967=1148.296,319.197,-75.759,-176.773,8.717,148.795
C04968=1148.300,318.949,-75.727,-176.776,8.713,148.794
C04969=1148.304,318.702,-75.695,-176.778,8.710,148.794
C04970=1148.309,318.453,-75.663,-176.781,8.706,148.794
C04971=1148.312,318.205,-75.631,-176.783,8.703,148.794
C04972=1148.316,317.958,-75.598,-176.785,8.700,148.794
C04973=1148.320,317.710,-75.566,-176.788,8.696,148.793
C04974=1148.325,317.462,-75.534,-176.791,8.692,148.793
C04975=1148.329,317.214,-75.502,-176.794,8.688,148.793
C04976=1148.333,316.966,-75.470,-176.796,8.685,148.793
C04977=1148.337,316.719,-75.439,-176.799,8.682,148.793
C04978=1148.342,316.470,-75.406,-176.802,8.678,148.792
C04979=1148.345,316.222,-75.374,-176.804,8.675,148.792
C04980=1148.350,315.974,-75.342,-176.806,8.671,148.792
C04981=1148.354,315.727,-75.310,-176.809,8.667,148.792
C04982=1148.357,315.479,-75.278,-176.812,8.664,148.792
C04983=1148.362,315.231,-75.245,-176.814,8.661,148.792
C04984=1148.366,314.983,-75.214,-176.817,8.657,148.791
C04985=1148.370,314.735,-75.182,-176.819,8.654,148.791
C04986=1148.374,314.487,-75.151,-176.822,8.650,148.791
C04987=1148.379,314.239,-75.119,-176.825,8.647,148.791
C04988=1148.383,313.991,-75.087,-176.827,8.643,148.791
C04989=1148.387,313.713,-75.052,-176.830,8.639,148.791
C04990=1148.392,313.436,-75.015,-176.833,8.635,148.790
C04991=1148.396,313.158,-74.980,-176.836,8.631,148.790
C04992=1148.401,312.881,-74.944,-176.839,8.628,148.790
C04993=1148.405,312.633,-74.913,-176.842,8.624,148.790
C04994=1148.409,312.385,-74.881,-176.844,8.621,148.790
C04995=1148.413,312.136,-74.849,-176.846,8.618,148.790
C04996=1148.418,311.889,-74.818,-176.849,8.613,148.789
C04997=1148.421,311.641,-74.786,-176.852,8.610,148.789
C04998=1148.426,311.393,-74.754,-176.854,8.607,148.789
C04999=1148.430,311.145,-74.723,-176.857,8.603,148.789
C05000=1148.434,310.896,-74.691,-176.860,8.600,148.789
C05001=1148.438,310.649,-74.659,-176.862,8.597,148.789
C05002=1148.442,310.401,-74.627,-176.865,8.593,148.789
C05003=1148.447,310.153,-74.597,-176.868,8.590,148.788
C05004=1148.450,309.905,-74.565,-176.870,8.586,148.788
C05005=1148.455,309.658,-74.533,-176.873,8.583,148.788
C05006=1148.459,309.409,-74.502,-176.876,8.579,148.788
C05007=1148.463,309.161,-74.470,-176.878,8.576,148.788
C05008=1148.468,308.913,-74.438,-176.880,8.573,148.788
C05009=1148.472,308.665,-74.407,-176.884,8.569,148.788
C05010=1148.476,308.417,-74.376,-176.886,8.566,148.788
C05011=1148.480,308.169,-74.344,-176.888,8.562,148.787
C05012=1148.484,307.921,-74.313,-176.891,8.558,148.787
C05013=1148.488,307.673,-74.281,-176.894,8.555,148.787
C05014=1148.493,307.425,-74.250,-176.896,8.552,148.787
C05015=1148.496,307.177,-74.219,-176.899,8.549,148.787
C05016=1148.501,306.929,-74.188,-176.902,8.545,148.787
C05017=1148.505,306.681,-74.156,-176.904,8.542,148.787
C05018=1148.509,306.433,-74.125,-176.907,8.539,148.786
C05019=1148.513,306.185,-74.093,-176.910,8.534,148.786
C05020=1148.517,305.937,-74.063,-176.912,8.532,148.786
C05021=1148.521,305.689,-74.031,-176.915,8.528,148.786
C05022=1148.526,305.441,-74.000,-176.917,8.525,148.786
C05023=1148.529,305.193,-73.968,-176.920,8.521,148.786
C05024=1148.534,304.945,-73.937,-176.923,8.518,148.786
C05025=1148.538,304.697,-73.906,-176.925,8.515,148.786
C05026=1148.542,304.449,-73.875,-176.928,8.511,148.785
C05027=1148.547,304.201,-73.844,-176.931,8.508,148.785
C05028=1148.551,303.953,-73.812,-176.933,8.504,148.785
C05029=1148.555,303.705,-73.781,-176.936,8.501,148.785
C05030=1148.559,303.457,-73.750,-176.939,8.497,148.785
C05031=1148.564,303.209,-73.719,-176.941,8.494,148.785
C05032=1148.568,302.961,-73.688,-176.944,8.491,148.785
C05033=1148.572,302.713,-73.657,-176.946,8.488,148.785
C05034=1148.576,302.465,-73.627,-176.949,8.484,148.784
C05035=1148.580,302.217,-73.595,-176.952,8.481,148.784
C05036=1148.585,301.969,-73.564,-176.954,8.478,148.784
C05037=1148.589,301.721,-73.533,-176.956,8.474,148.784
C05038=1148.593,301.473,-73.502,-176.960,8.471,148.784
C05039=1148.597,301.225,-73.471,-176.962,8.467,148.784
C05040=1148.601,300.977,-73.440,-176.965,8.464,148.784
C05041=1148.605,300.729,-73.409,-176.967,8.461,148.784
C05042=1148.610,300.481,-73.379,-176.970,8.457,148.784
C05043=1148.614,300.232,-73.348,-176.973,8.454,148.784
C05044=1148.619,299.984,-73.317,-176.975,8.451,148.783
C05045=1148.622,299.737,-73.285,-176.978,8.447,148.783
C05046=1148.626,299.489,-73.255,-176.981,8.444,148.783
C05047=1148.631,299.241,-73.224,-176.983,8.440,148.783
C05048=1148.635,298.992,-73.193,-176.986,8.437,148.783
C05049=1148.639,298.744,-73.163,-176.988,8.434,148.783
C05050=1148.643,298.496,-73.132,-176.991,8.430,148.783
C05051=1148.647,298.248,-73.101,-176.994,8.427,148.783
C05052=1148.651,298.000,-73.071,-176.996,8.424,148.783
C05053=1148.656,297.752,-73.040,-176.999,8.421,148.783
C05054=1148.660,297.504,-73.009,-177.002,8.417,148.782
C05055=1148.664,297.256,-72.978,-177.005,8.414,148.782
C05056=1148.668,297.008,-72.948,-177.007,8.411,148.782
C05057=1148.673,296.760,-72.917,-177.009,8.407,148.782
C05058=1148.677,296.511,-72.886,-177.012,8.404,148.782
C05059=1148.681,296.264,-72.856,-177.015,8.400,148.782
C05060=1148.685,296.016,-72.825,-177.018,8.397,148.782
C05061=1148.689,295.768,-72.795,-177.020,8.394,148.782
C05062=1148.694,295.519,-72.764,-177.023,8.391,148.782
C05063=1148.698,295.271,-72.734,-177.026,8.387,148.782
C05064=1148.702,295.023,-72.703,-177.029,8.384,148.782
C05065=1148.707,294.775,-72.673,-177.031,8.381,148.781
C05066=1148.710,294.527,-72.642,-177.034,8.378,148.781
C05067=1148.715,294.279,-72.611,-177.036,8.375,148.781
C05068=1148.719,294.031,-72.582,-177.039,8.371,148.781
C05069=1148.723,293.783,-72.551,-177.042,8.368,148.781
C05070=1148.727,293.534,-72.521,-177.044,8.364,148.781
C05071=1148.731,293.286,-72.490,-177.047,8.361,148.781
C05072=1148.736,293.038,-72.459,-177.049,8.358,148.781
C05073=1148.740,292.790,-72.430,-177.052,8.354,148.781
C05074=1148.745,292.542,-72.399,-177.055,8.351,148.781
C05075=1148.748,292.294,-72.368,-177.058,8.348,148.781
C05076=1148.753,292.045,-72.338,-177.060,8.345,148.780
C05077=1148.757,291.798,-72.308,-177.063,8.342,148.781
C05078=1148.761,291.550,-72.278,-177.066,8.338,148.780
C05079=1148.766,291.301,-72.248,-177.068,8.335,148.780
C05080=1148.769,291.053,-72.217,-177.071,8.332,148.780
C05081=1148.773,290.805,-72.187,-177.073,8.329,148.780
C05082=1148.778,290.557,-72.157,-177.076,8.326,148.780
C05083=1148.782,290.309,-72.126,-177.079,8.322,148.780
C05084=1148.786,290.061,-72.097,-177.082,8.319,148.780
C05085=1148.790,289.813,-72.067,-177.084,8.316,148.780
C05086=1148.795,289.564,-72.037,-177.087,8.313,148.780
C05087=1148.798,289.316,-72.006,-177.089,8.309,148.780
C05088=1148.803,289.068,-71.975,-177.092,8.306,148.780
C05089=1148.807,288.820,-71.946,-177.095,8.302,148.780
C05090=1148.811,288.572,-71.916,-177.098,8.299,148.780
C05091=1148.816,288.324,-71.886,-177.100,8.296,148.779
C05092=1148.820,288.075,-71.856,-177.103,8.293,148.780
C05093=1148.825,287.801,-71.823,-177.106,8.289,148.780
C05094=1148.830,287.525,-71.789,-177.109,8.286,148.779
C05095=1148.835,287.249,-71.756,-177.112,8.282,148.779
C05096=1148.839,286.975,-71.723,-177.115,8.278,148.779
C05097=1148.843,286.726,-71.693,-177.118,8.275,148.779
C05098=1148.847,286.478,-71.663,-177.120,8.272,148.779
C05099=1148.852,286.229,-71.633,-177.123,8.269,148.779
C05100=1148.856,285.981,-71.603,-177.125,8.266,148.779
C05101=1148.860,285.733,-71.573,-177.128,8.263,148.779
C05102=1148.865,285.485,-71.543,-177.131,8.259,148.779
C05103=1148.869,285.237,-71.514,-177.133,8.256,148.779
C05104=1148.873,284.989,-71.483,-177.136,8.253,148.779
C05105=1148.877,284.741,-71.454,-177.139,8.250,148.779
C05106=1148.882,284.492,-71.424,-177.141,8.247,148.779
C05107=1148.886,284.244,-71.395,-177.144,8.244,148.779
C05108=1148.890,283.996,-71.364,-177.147,8.241,148.779
C05109=1148.894,283.748,-71.335,-177.150,8.237,148.779
C05110=1148.898,283.500,-71.305,-177.153,8.234,148.779
C05111=1148.902,283.251,-71.276,-177.155,8.231,148.778
C05112=1148.907,283.003,-71.246,-177.158,8.228,148.779
C05113=1148.911,282.755,-71.216,-177.160,8.225,148.779
C05114=1148.915,282.507,-71.186,-177.163,8.221,148.778
C05115=1148.919,282.259,-71.157,-177.165,8.218,148.778
C05116=1148.924,282.010,-71.127,-177.169,8.215,148.778
C05117=1148.928,281.762,-71.098,-177.171,8.211,148.778
C05118=1148.933,281.514,-71.068,-177.174,8.208,148.778
C05119=1148.937,281.265,-71.038,-177.176,8.205,148.778
C05120=1148.942,281.018,-71.009,-177.179,8.202,148.778
C05121=1148.946,280.769,-70.980,-177.182,8.199,148.778
C05122=1148.950,280.521,-70.950,-177.184,8.196,148.778
C05123=1148.954,280.273,-70.921,-177.187,8.193,148.778
C05124=1148.958,280.025,-70.892,-177.190,8.189,148.778
C05125=1148.963,279.776,-70.862,-177.193,8.186,148.778
C05126=1148.967,279.528,-70.833,-177.195,8.183,148.778
C05127=1148.971,279.280,-70.803,-177.198,8.180,148.778
C05128=1148.975,279.032,-70.774,-177.200,8.177,148.778
C05129=1148.979,278.783,-70.744,-177.203,8.174,148.778
C05130=1148.984,278.535,-70.715,-177.206,8.171,148.778
C05131=1148.988,278.287,-70.686,-177.208,8.168,148.778
C05132=1148.993,278.039,-70.656,-177.211,8.165,148.778
C05133=1148.997,277.791,-70.627,-177.214,8.161,148.778
C05134=1149.001,277.543,-70.597,-177.217,8.158,148.778
C05135=1149.005,277.294,-70.568,-177.220,8.155,148.778
C05136=1149.010,277.046,-70.539,-177.222,8.152,148.778
C05137=1149.014,276.797,-70.510,-177.225,8.149,148.778
C05138=1149.018,276.549,-70.480,-177.227,8.146,148.778
C05139=1149.023,276.301,-70.451,-177.230,8.143,148.778
C05140=1149.027,276.053,-70.422,-177.233,8.140,148.778
C05141=1149.031,275.804,-70.393,-177.235,8.137,148.778
C05142=1149.035,275.556,-70.364,-177.238,8.134,148.778
C05143=1149.039,275.308,-70.335,-177.241,8.130,148.778
C05144=1149.043,275.060,-70.305,-177.244,8.127,148.778
C05145=1149.048,274.812,-70.277,-177.247,8.124,148.778
C05146=1149.052,274.563,-70.247,-177.249,8.121,148.778
C05147=1149.057,274.315,-70.218,-177.252,8.118,148.778
C05148=1149.061,274.067,-70.188,-177.255,8.115,148.778
C05149=1149.065,273.818,-70.160,-177.257,8.112,148.778
C05150=1149.069,273.571,-70.131,-177.260,8.109,148.778
C05151=1149.074,273.322,-70.102,-177.263,8.106,148.778
C05152=1149.078,273.074,-70.073,-177.266,8.103,148.778
C05153=1149.082,272.825,-70.044,-177.268,8.100,148.778
C05154=1149.087,272.577,-70.015,-177.271,8.097,148.778
C05155=1149.091,272.329,-69.986,-177.273,8.094,148.778
C05156=1149.095,272.081,-69.957,-177.277,8.090,148.778
C05157=1149.099,271.832,-69.928,-177.279,8.087,148.778
C05158=1149.104,271.584,-69.899,-177.282,8.084,148.778
C05159=1149.108,271.336,-69.871,-177.285,8.081,148.778
C05160=1149.112,271.088,-69.842,-177.287,8.078,148.778
C05161=1149.117,270.839,-69.813,-177.290,8.075,148.778
C05162=1149.121,270.591,-69.784,-177.293,8.072,148.778
C05163=1149.125,270.342,-69.756,-177.295,8.069,148.778
C05164=1149.129,270.094,-69.726,-177.298,8.066,148.778
C05165=1149.134,269.846,-69.698,-177.301,8.063,148.778
C05166=1149.138,269.597,-69.670,-177.303,8.060,148.778
C05167=1149.142,269.349,-69.640,-177.306,8.057,148.778
C05168=1149.147,269.101,-69.612,-177.309,8.054,148.778
C05169=1149.151,268.853,-69.583,-177.312,8.051,148.778
C05170=1149.155,268.604,-69.554,-177.314,8.047,148.778
C05171=1149.160,268.356,-69.526,-177.317,8.045,148.778
C05172=1149.164,268.108,-69.497,-177.319,8.042,148.778
C05173=1149.168,267.859,-69.468,-177.323,8.038,148.778
C05174=1149.173,267.611,-69.440,-177.326,8.035,148.778
C05175=1149.177,267.363,-69.411,-177.328,8.032,148.778
C05176=1149.181,267.114,-69.382,-177.331,8.029,148.778
C05177=1149.186,266.866,-69.354,-177.333,8.026,148.778
C05178=1149.190,266.618,-69.325,-177.336,8.023,148.778
C05179=1149.194,266.369,-69.296,-177.339,8.020,148.778
C05180=1149.199,266.121,-69.268,-177.342,8.017,148.778
C05181=1149.203,265.872,-69.240,-177.345,8.014,148.778
C05182=1149.207,265.625,-69.211,-177.347,8.011,148.778
C05183=1149.212,265.376,-69.183,-177.350,8.008,148.778
C05184=1149.216,265.128,-69.154,-177.352,8.005,148.778
C05185=1149.221,264.879,-69.126,-177.355,8.002,148.778
C05186=1149.224,264.631,-69.098,-177.358,7.999,148.778
C05187=1149.229,264.383,-69.069,-177.361,7.996,148.778
C05188=1149.233,264.135,-69.041,-177.363,7.993,148.778
C05189=1149.238,263.887,-69.012,-177.366,7.990,148.778
C05190=1149.242,263.638,-68.984,-177.369,7.987,148.778
C05191=1149.247,263.390,-68.956,-177.371,7.984,148.778
C05192=1149.251,263.141,-68.928,-177.374,7.981,148.778
C05193=1149.255,262.892,-68.899,-177.377,7.978,148.778
C05194=1149.259,262.644,-68.871,-177.380,7.975,148.778
C05195=1149.264,262.396,-68.842,-177.382,7.972,148.778
C05196=1149.268,262.148,-68.815,-177.385,7.969,148.778
C05197=1149.273,261.874,-68.784,-177.388,7.965,148.778
C05198=1149.278,261.601,-68.752,-177.391,7.962,148.778
C05199=1149.282,261.327,-68.721,-177.394,7.959,148.778
C05200=1149.287,261.054,-68.690,-177.397,7.956,148.778
C05201=1149.292,260.806,-68.662,-177.400,7.953,148.779
C05202=1149.296,260.557,-68.634,-177.403,7.950,148.779
C05203=1149.300,260.309,-68.606,-177.405,7.947,148.779
C05204=1149.304,260.060,-68.577,-177.408,7.944,148.779
C05205=1149.309,259.813,-68.549,-177.411,7.941,148.779
C05206=1149.313,259.563,-68.522,-177.414,7.938,148.779
C05207=1149.318,259.315,-68.494,-177.417,7.935,148.779
C05208=1149.322,259.067,-68.465,-177.419,7.932,148.779
C05209=1149.326,258.819,-68.438,-177.422,7.929,148.779
C05210=1149.331,258.570,-68.409,-177.424,7.926,148.779
C05211=1149.335,258.322,-68.381,-177.427,7.923,148.779
C05212=1149.339,258.073,-68.354,-177.430,7.920,148.779
C05213=1149.343,257.825,-68.326,-177.433,7.917,148.779
C05214=1149.348,257.577,-68.298,-177.436,7.914,148.779
C05215=1149.352,257.328,-68.269,-177.438,7.911,148.779
C05216=1149.357,257.080,-68.242,-177.441,7.908,148.779
C05217=1149.361,256.832,-68.215,-177.443,7.906,148.779
C05218=1149.366,256.583,-68.186,-177.446,7.903,148.779
C05219=1149.370,256.335,-68.158,-177.449,7.900,148.779
C05220=1149.374,256.086,-68.131,-177.452,7.897,148.780
C05221=1149.378,255.838,-68.103,-177.454,7.895,148.780
C05222=1149.383,255.590,-68.074,-177.457,7.891,148.779
C05223=1149.387,255.340,-68.047,-177.460,7.888,148.780
C05224=1149.392,255.093,-68.019,-177.462,7.885,148.780
C05225=1149.396,254.844,-67.991,-177.465,7.882,148.780
C05226=1149.400,254.596,-67.964,-177.468,7.880,148.780
C05227=1149.405,254.348,-67.936,-177.471,7.877,148.780
C05228=1149.409,254.098,-67.908,-177.473,7.874,148.780
C05229=1149.414,253.850,-67.880,-177.476,7.871,148.780
C05230=1149.418,253.602,-67.853,-177.479,7.868,148.780
C05231=1149.422,253.353,-67.825,-177.482,7.865,148.780
C05232=1149.426,253.105,-67.798,-177.485,7.862,148.780
C05233=1149.431,252.857,-67.770,-177.487,7.859,148.780
C05234=1149.435,252.608,-67.742,-177.490,7.856,148.780
C05235=1149.440,252.360,-67.715,-177.493,7.853,148.780
C05236=1149.444,252.112,-67.687,-177.496,7.850,148.780
C05237=1149.448,251.863,-67.660,-177.499,7.847,148.780
C05238=1149.452,251.615,-67.632,-177.501,7.844,148.781
C05239=1149.457,251.366,-67.605,-177.504,7.841,148.781
C05240=1149.462,251.118,-67.578,-177.506,7.839,148.781
C05241=1149.466,250.869,-67.549,-177.509,7.836,148.781
C05242=1149.471,250.620,-67.522,-177.512,7.833,148.781
C05243=1149.475,250.373,-67.495,-177.515,7.831,148.781
C05244=1149.479,250.123,-67.467,-177.517,7.828,148.781
C05245=1149.484,249.875,-67.440,-177.520,7.825,148.781
C05246=1149.488,249.627,-67.412,-177.523,7.822,148.781
C05247=1149.492,249.379,-67.386,-177.526,7.819,148.781
C05248=1149.496,249.130,-67.358,-177.529,7.816,148.781
C05249=1149.501,248.882,-67.331,-177.531,7.813,148.781
C05250=1149.505,248.633,-67.304,-177.534,7.810,148.781
C05251=1149.510,248.385,-67.277,-177.537,7.807,148.781
C05252=1149.514,248.136,-67.249,-177.540,7.804,148.782
C05253=1149.518,247.888,-67.221,-177.542,7.802,148.782
C05254=1149.523,247.639,-67.194,-177.545,7.799,148.782
C05255=1149.528,247.391,-67.167,-177.547,7.796,148.782
C05256=1149.532,247.142,-67.140,-177.550,7.793,148.782
C05257=1149.536,246.894,-67.112,-177.553,7.790,148.782
C05258=1149.541,246.645,-67.085,-177.556,7.787,148.782
C05259=1149.545,246.397,-67.058,-177.559,7.784,148.782
C05260=1149.549,246.148,-67.031,-177.561,7.782,148.782
C05261=1149.554,245.900,-67.004,-177.565,7.779,148.782
C05262=1149.558,245.651,-66.977,-177.567,7.776,148.783
C05263=1149.563,245.402,-66.950,-177.570,7.773,148.783
C05264=1149.567,245.154,-66.922,-177.572,7.771,148.783
C05265=1149.572,244.906,-66.895,-177.575,7.768,148.783
C05266=1149.575,244.658,-66.869,-177.578,7.765,148.783
C05267=1149.580,244.409,-66.841,-177.581,7.762,148.783
C05268=1149.585,244.161,-66.814,-177.584,7.759,148.783
C05269=1149.589,243.911,-66.787,-177.586,7.756,148.783
C05270=1149.593,243.663,-66.761,-177.589,7.753,148.783
C05271=1149.597,243.415,-66.733,-177.592,7.750,148.783
C05272=1149.602,243.166,-66.706,-177.595,7.748,148.783
C05273=1149.607,242.918,-66.679,-177.597,7.745,148.783
C05274=1149.611,242.670,-66.653,-177.600,7.742,148.783
C05275=1149.615,242.421,-66.626,-177.602,7.740,148.784
C05276=1149.620,242.173,-66.599,-177.606,7.737,148.784
C05277=1149.625,241.924,-66.572,-177.608,7.734,148.784
C05278=1149.628,241.675,-66.545,-177.611,7.731,148.784
C05279=1149.633,241.427,-66.518,-177.614,7.728,148.784
C05280=1149.638,241.178,-66.491,-177.617,7.725,148.784
C05281=1149.641,240.929,-66.465,-177.619,7.723,148.784
C05282=1149.646,240.681,-66.438,-177.622,7.720,148.784
C05283=1149.651,240.432,-66.411,-177.625,7.717,148.784
C05284=1149.655,240.184,-66.384,-177.627,7.714,148.784
C05285=1149.659,239.936,-66.357,-177.630,7.711,148.785
C05286=1149.664,239.687,-66.330,-177.633,7.709,148.785
C05287=1149.668,239.439,-66.305,-177.636,7.706,148.785
C05288=1149.673,239.190,-66.277,-177.638,7.704,148.785
C05289=1149.678,238.942,-66.250,-177.641,7.701,148.785
C05290=1149.681,238.693,-66.224,-177.644,7.698,148.785
C05291=1149.686,238.444,-66.198,-177.647,7.695,148.785
C05292=1149.690,238.196,-66.171,-177.650,7.692,148.785
C05293=1149.695,237.948,-66.144,-177.652,7.689,148.785
C05294=1149.699,237.699,-66.118,-177.656,7.687,148.786
C05295=1149.704,237.450,-66.091,-177.658,7.684,148.786
C05296=1149.709,237.202,-66.064,-177.661,7.682,148.786
C05297=1149.712,236.954,-66.038,-177.663,7.679,148.786
C05298=1149.717,236.704,-66.011,-177.666,7.676,148.786
C05299=1149.721,236.456,-65.985,-177.669,7.673,148.786
C05300=1149.726,236.207,-65.959,-177.672,7.670,148.786
C05301=1149.731,235.936,-65.930,-177.675,7.667,148.787
C05302=1149.736,235.664,-65.900,-177.678,7.664,148.787
C05303=1149.741,235.391,-65.871,-177.681,7.661,148.787
C05304=1149.745,235.120,-65.843,-177.683,7.658,148.787
C05305=1149.750,234.872,-65.816,-177.687,7.656,148.787
C05306=1149.754,234.623,-65.790,-177.689,7.653,148.787
C05307=1149.758,234.375,-65.763,-177.692,7.650,148.787
C05308=1149.763,234.126,-65.737,-177.695,7.647,148.787
C05309=1149.767,233.878,-65.711,-177.698,7.644,148.787
C05310=1149.772,233.629,-65.685,-177.700,7.642,148.787
C05311=1149.776,233.381,-65.658,-177.703,7.639,148.788
C05312=1149.781,233.132,-65.632,-177.706,7.637,148.788
C05313=1149.785,232.883,-65.605,-177.709,7.634,148.788
C05314=1149.789,232.635,-65.580,-177.712,7.631,148.788
C05315=1149.794,232.385,-65.553,-177.714,7.629,148.788
C05316=1149.798,232.137,-65.527,-177.717,7.626,148.788
C05317=1149.802,231.888,-65.501,-177.720,7.623,148.789
C05318=1149.808,231.641,-65.474,-177.723,7.620,148.789
C05319=1149.812,231.392,-65.449,-177.725,7.617,148.789
C05320=1149.817,231.143,-65.422,-177.728,7.615,148.789
C05321=1149.821,230.895,-65.396,-177.730,7.612,148.789
C05322=1149.825,230.646,-65.370,-177.734,7.610,148.789
C05323=1149.830,230.397,-65.344,-177.736,7.607,148.789
C05324=1149.834,230.148,-65.317,-177.739,7.604,148.789
C05325=1149.839,229.900,-65.292,-177.741,7.602,148.789
C05326=1149.843,229.652,-65.266,-177.744,7.599,148.790
C05327=1149.848,229.402,-65.240,-177.747,7.596,148.790
C05328=1149.852,229.154,-65.213,-177.750,7.593,148.790
C05329=1149.856,228.905,-65.188,-177.753,7.590,148.790
C05330=1149.861,228.657,-65.162,-177.755,7.588,148.790
C05331=1149.866,228.408,-65.136,-177.758,7.585,148.790
C05332=1149.870,228.160,-65.109,-177.761,7.583,148.791
C05333=1149.874,227.911,-65.084,-177.764,7.580,148.791
C05334=1149.878,227.662,-65.058,-177.766,7.578,148.791
C05335=1149.884,227.414,-65.032,-177.769,7.575,148.791
C05336=1149.888,227.165,-65.006,-177.772,7.572,148.791
C05337=1149.892,226.916,-64.980,-177.775,7.569,148.791
C05338=1149.896,226.668,-64.954,-177.777,7.567,148.791
C05339=1149.901,226.420,-64.928,-177.780,7.564,148.791
C05340=1149.906,226.171,-64.902,-177.783,7.562,148.792
C05341=1149.910,225.922,-64.876,-177.786,7.559,148.792
C05342=1149.914,225.673,-64.851,-177.788,7.557,148.792
C05343=1149.919,225.425,-64.825,-177.791,7.554,148.792
C05344=1149.923,225.176,-64.799,-177.794,7.551,148.792
C05345=1149.928,224.928,-64.774,-177.797,7.548,148.792
C05346=1149.932,224.679,-64.748,-177.800,7.545,148.792
C05347=1149.937,224.431,-64.723,-177.802,7.543,148.793
C05348=1149.942,224.182,-64.696,-177.805,7.541,148.793
C05349=1149.946,223.933,-64.671,-177.808,7.538,148.793
C05350=1149.951,223.685,-64.645,-177.810,7.535,148.793
C05351=1149.955,223.436,-64.619,-177.813,7.533,148.793
C05352=1149.959,223.187,-64.594,-177.816,7.530,148.794
C05353=1149.963,222.938,-64.568,-177.819,7.527,148.794
C05354=1149.968,222.690,-64.542,-177.821,7.525,148.794
C05355=1149.972,222.441,-64.517,-177.824,7.522,148.794
C05356=1149.977,222.193,-64.491,-177.827,7.519,148.794
C05357=1149.982,221.944,-64.466,-177.830,7.517,148.794
C05358=1149.986,221.695,-64.441,-177.832,7.514,148.794
C05359=1149.990,221.446,-64.415,-177.836,7.512,148.795
C05360=1149.995,221.198,-64.389,-177.839,7.509,148.795
C05361=1149.999,220.949,-64.364,-177.841,7.506,148.795
C05362=1150.004,220.701,-64.338,-177.844,7.504,148.795
C05363=1150.009,220.452,-64.313,-177.847,7.501,148.795
C05364=1150.013,220.203,-64.288,-177.850,7.498,148.795
C05365=1150.018,219.955,-64.262,-177.852,7.496,148.795
C05366=1150.022,219.706,-64.236,-177.855,7.494,148.796
C05367=1150.026,219.457,-64.211,-177.858,7.491,148.796
C05368=1150.031,219.209,-64.186,-177.861,7.488,148.796
C05369=1150.036,218.960,-64.160,-177.863,7.486,148.796
C05370=1150.040,218.712,-64.135,-177.866,7.483,148.796
C05371=1150.044,218.463,-64.110,-177.869,7.480,148.796
C05372=1150.048,218.214,-64.085,-177.871,7.478,148.797
C05373=1150.053,217.966,-64.059,-177.874,7.476,148.797
C05374=1150.058,217.716,-64.034,-177.877,7.473,148.797
C05375=1150.063,217.468,-64.009,-177.879,7.471,148.797
C05376=1150.067,217.219,-63.983,-177.883,7.468,148.797
C05377=1150.072,216.971,-63.958,-177.885,7.465,148.798
C05378=1150.075,216.722,-63.933,-177.888,7.463,148.798
C05379=1150.080,216.473,-63.907,-177.891,7.460,148.798
C05380=1150.085,216.225,-63.883,-177.894,7.457,148.798
C05381=1150.089,215.976,-63.857,-177.896,7.455,148.798
C05382=1150.094,215.727,-63.832,-177.899,7.453,148.799
C05383=1150.098,215.478,-63.807,-177.902,7.450,148.799
C05384=1150.103,215.230,-63.783,-177.905,7.447,148.799
C05385=1150.107,214.981,-63.757,-177.907,7.445,148.799
C05386=1150.112,214.732,-63.732,-177.910,7.442,148.799
C05387=1150.116,214.484,-63.706,-177.913,7.439,148.799
C05388=1150.121,214.235,-63.682,-177.916,7.438,148.800
C05389=1150.125,213.986,-63.657,-177.918,7.435,148.800
C05390=1150.130,213.738,-63.632,-177.921,7.432,148.800
C05391=1150.134,213.489,-63.606,-177.924,7.430,148.800
C05392=1150.139,213.240,-63.582,-177.927,7.427,148.800
C05393=1150.143,212.991,-63.557,-177.929,7.425,148.801
C05394=1150.148,212.743,-63.532,-177.932,7.422,148.801
C05395=1150.152,212.494,-63.507,-177.935,7.419,148.801
C05396=1150.157,212.246,-63.482,-177.938,7.418,148.801
C05397=1150.162,211.997,-63.457,-177.940,7.415,148.801
C05398=1150.166,211.747,-63.432,-177.943,7.412,148.801
C05399=1150.170,211.500,-63.407,-177.946,7.410,148.802
C05400=1150.175,211.250,-63.382,-177.949,7.407,148.802
C05401=1150.180,211.002,-63.358,-177.952,7.405,148.802
C05402=1150.184,210.753,-63.332,-177.954,7.403,148.802
C05403=1150.189,210.504,-63.308,-177.957,7.400,148.802
C05404=1150.193,210.256,-63.284,-177.960,7.397,148.803
C05405=1150.198,209.985,-63.256,-177.963,7.394,148.803
C05406=1150.203,209.714,-63.229,-177.966,7.392,148.803
C05407=1150.208,209.444,-63.202,-177.969,7.389,148.803
C05408=1150.213,209.174,-63.176,-177.972,7.387,148.803
C05409=1150.217,208.924,-63.151,-177.975,7.384,148.804
C05410=1150.222,208.676,-63.126,-177.978,7.381,148.804
C05411=1150.226,208.427,-63.101,-177.980,7.379,148.804
C05412=1150.231,208.178,-63.077,-177.983,7.376,148.804
C05413=1150.236,207.930,-63.052,-177.986,7.375,148.804
C05414=1150.240,207.681,-63.028,-177.988,7.372,148.805
C05415=1150.245,207.432,-63.003,-177.992,7.369,148.805
C05416=1150.249,207.183,-62.979,-177.994,7.367,148.805
C05417=1150.253,206.935,-62.953,-177.997,7.364,148.805
C05418=1150.258,206.686,-62.929,-178.000,7.362,148.805
C05419=1150.263,206.438,-62.904,-178.002,7.359,148.806
C05420=1150.267,206.188,-62.880,-178.005,7.357,148.806
C05421=1150.272,205.940,-62.855,-178.008,7.355,148.806
C05422=1150.276,205.691,-62.831,-178.011,7.352,148.806
C05423=1150.281,205.442,-62.806,-178.014,7.349,148.806
C05424=1150.285,205.193,-62.782,-178.016,7.348,148.807
C05425=1150.290,204.945,-62.757,-178.019,7.345,148.807
C05426=1150.294,204.696,-62.733,-178.021,7.342,148.807
C05427=1150.299,204.447,-62.708,-178.025,7.340,148.807
C05428=1150.304,204.198,-62.684,-178.027,7.338,148.807
C05429=1150.308,203.950,-62.660,-178.030,7.335,148.808
C05430=1150.313,203.701,-62.635,-178.033,7.332,148.808
C05431=1150.317,203.452,-62.611,-178.036,7.331,148.808
C05432=1150.322,203.204,-62.586,-178.038,7.328,148.808
C05433=1150.326,202.954,-62.563,-178.041,7.326,148.809
C05434=1150.331,202.705,-62.538,-178.044,7.323,148.809
C05435=1150.336,202.457,-62.514,-178.047,7.320,148.809
C05436=1150.340,202.208,-62.490,-178.049,7.318,148.809
C05437=1150.344,201.959,-62.465,-178.052,7.315,148.809
C05438=1150.349,201.710,-62.441,-178.055,7.314,148.810
C05439=1150.353,201.462,-62.417,-178.058,7.311,148.810
C05440=1150.358,201.213,-62.393,-178.060,7.309,148.810
C05441=1150.363,200.964,-62.369,-178.063,7.306,148.810
C05442=1150.367,200.715,-62.344,-178.066,7.304,148.811
C05443=1150.371,200.467,-62.320,-178.069,7.301,148.811
C05444=1150.376,200.218,-62.296,-178.072,7.299,148.811
C05445=1150.381,199.969,-62.272,-178.074,7.297,148.811
C05446=1150.386,199.721,-62.248,-178.077,7.294,148.811
C05447=1150.389,199.471,-62.223,-178.079,7.292,148.812
C05448=1150.395,199.223,-62.199,-178.083,7.290,148.812
C05449=1150.399,198.974,-62.175,-178.085,7.287,148.812
C05450=1150.404,198.725,-62.151,-178.088,7.285,148.812
C05451=1150.408,198.477,-62.127,-178.090,7.283,148.813
C05452=1150.412,198.227,-62.104,-178.094,7.280,148.813
C05453=1150.417,197.978,-62.079,-178.097,7.277,148.813
C05454=1150.422,197.730,-62.055,-178.099,7.276,148.813
C05455=1150.426,197.481,-62.031,-178.102,7.273,148.813
C05456=1150.431,197.233,-62.007,-178.105,7.271,148.814
C05457=1150.436,196.983,-61.984,-178.107,7.268,148.814
C05458=1150.441,196.735,-61.959,-178.110,7.266,148.814
C05459=1150.444,196.486,-61.935,-178.113,7.263,148.814
C05460=1150.449,196.237,-61.912,-178.116,7.262,148.815
C05461=1150.454,195.988,-61.887,-178.118,7.259,148.815
C05462=1150.458,195.739,-61.864,-178.121,7.257,148.815
C05463=1150.463,195.491,-61.840,-178.124,7.254,148.815
C05464=1150.467,195.242,-61.817,-178.127,7.252,148.816
C05465=1150.472,194.993,-61.792,-178.130,7.250,148.816
C05466=1150.477,194.744,-61.769,-178.132,7.248,148.816
C05467=1150.482,194.496,-61.745,-178.135,7.245,148.816
C05468=1150.486,194.247,-61.721,-178.138,7.243,148.817
C05469=1150.490,193.997,-61.697,-178.141,7.240,148.817
C05470=1150.495,193.748,-61.673,-178.143,7.238,148.817
C05471=1150.499,193.500,-61.649,-178.146,7.236,148.817
C05472=1150.504,193.251,-61.626,-178.149,7.234,148.817
C05473=1150.509,193.002,-61.603,-178.152,7.231,148.818
C05474=1150.513,192.753,-61.579,-178.155,7.229,148.818
C05475=1150.518,192.504,-61.555,-178.157,7.226,148.818
C05476=1150.522,192.256,-61.531,-178.160,7.225,148.819
C05477=1150.527,192.007,-61.508,-178.163,7.222,148.819
C05478=1150.531,191.758,-61.484,-178.165,7.220,148.819
C05479=1150.536,191.510,-61.460,-178.168,7.217,148.819
